C03654=1194.031,57.850,-47.386,-179.235,5.821,148.807
C03655=1194.026,58.099,-47.403,-179.232,5.823,148.806
C03656=1194.021,58.349,-47.419,-179.230,5.824,148.805
C03657=1194.016,58.598,-47.436,-179.227,5.824,148.805
C03658=1194.011,58.848,-47.452,-179.225,5.825,148.804
C03659=1194.006,59.097,-47.468,-179.223,5.826,148.804
C03660=1194.001,59.346,-47.485,-179.219,5.827,148.803
C03661=1193.997,59.596,-47.502,-179.217,5.828,148.803
C03662=1193.992,59.844,-47.518,-179.215,5.828,148.802
C03663=1193.986,60.095,-47.535,-179.212,5.829,148.801
C03664=1193.981,60.344,-47.551,-179.209,5.831,148.801
C03665=1193.976,60.593,-47.568,-179.207,5.831,148.800
C03666=1193.972,60.843,-47.584,-179.204,5.832,148.800
C03667=1193.966,61.092,-47.601,-179.202,5.833,148.799
C03668=1193.962,61.341,-47.618,-179.199,5.833,148.798
C03669=1193.957,61.591,-47.634,-179.196,5.834,148.798
C03670=1193.952,61.840,-47.650,-179.194,5.835,148.797
C03671=1193.947,62.090,-47.667,-179.191,5.836,148.797
C03672=1193.942,62.339,-47.684,-179.189,5.836,148.796
C03673=1193.937,62.588,-47.700,-179.186,5.838,148.796
C03674=1193.932,62.838,-47.718,-179.183,5.839,148.795
C03675=1193.927,63.087,-47.734,-179.181,5.840,148.794
C03676=1193.922,63.336,-47.751,-179.178,5.840,148.794
C03677=1193.918,63.586,-47.767,-179.176,5.841,148.793
C03678=1193.913,63.836,-47.784,-179.173,5.842,148.793
C03679=1193.907,64.084,-47.801,-179.170,5.843,148.792
C03680=1193.903,64.334,-47.817,-179.168,5.843,148.791
C03681=1193.897,64.584,-47.834,-179.166,5.844,148.791
C03682=1193.892,64.833,-47.850,-179.162,5.846,148.790
C03683=1193.887,65.083,-47.868,-179.160,5.847,148.790
C03684=1193.883,65.332,-47.884,-179.158,5.847,148.789
C03685=1193.878,65.581,-47.901,-179.155,5.848,148.789
C03686=1193.872,65.831,-47.918,-179.152,5.849,148.788
C03687=1193.868,66.080,-47.934,-179.150,5.850,148.787
C03688=1193.864,66.329,-47.952,-179.147,5.851,148.787
C03689=1193.858,66.578,-47.969,-179.145,5.851,148.786
C03690=1193.853,66.828,-47.985,-179.142,5.853,148.786
C03691=1193.848,67.078,-48.003,-179.140,5.854,148.785
C03692=1193.843,67.326,-48.019,-179.137,5.854,148.785
C03693=1193.839,67.576,-48.036,-179.134,5.855,148.784
C03694=1193.833,67.826,-48.053,-179.132,5.856,148.784
C03695=1193.829,68.075,-48.070,-179.129,5.857,148.783
C03696=1193.823,68.324,-48.086,-179.126,5.858,148.782
C03697=1193.819,68.574,-48.103,-179.124,5.858,148.782
C03698=1193.813,68.823,-48.120,-179.121,5.860,148.781
C03699=1193.809,69.072,-48.138,-179.119,5.861,148.781
C03700=1193.804,69.322,-48.155,-179.116,5.861,148.780
C03701=1193.799,69.571,-48.171,-179.113,5.863,148.779
C03702=1193.794,69.820,-48.188,-179.111,5.864,148.779
C03703=1193.789,70.070,-48.205,-179.108,5.864,148.778
C03704=1193.785,70.320,-48.222,-179.106,5.865,148.778
C03705=1193.779,70.568,-48.240,-179.103,5.866,148.777
C03706=1193.775,70.818,-48.256,-179.100,5.867,148.777
C03707=1193.770,71.067,-48.274,-179.098,5.868,148.776
C03708=1193.765,71.317,-48.290,-179.095,5.868,148.775
C03709=1193.760,71.567,-48.307,-179.093,5.870,148.775
C03710=1193.754,71.815,-48.325,-179.090,5.871,148.774
C03711=1193.750,72.065,-48.342,-179.087,5.871,148.774
C03712=1193.745,72.314,-48.359,-179.085,5.873,148.773
C03713=1193.740,72.564,-48.376,-179.082,5.873,148.773
C03714=1193.735,72.813,-48.394,-179.080,5.874,148.772
C03715=1193.731,73.063,-48.410,-179.077,5.875,148.771
C03716=1193.725,73.312,-48.427,-179.074,5.876,148.771
C03717=1193.721,73.561,-48.445,-179.072,5.877,148.770
C03718=1193.716,73.810,-48.462,-179.069,5.878,148.770
C03719=1193.710,74.060,-48.479,-179.067,5.879,148.769
C03720=1193.706,74.310,-48.496,-179.064,5.880,148.769
C03721=1193.701,74.559,-48.514,-179.061,5.880,148.768
C03722=1193.696,74.808,-48.530,-179.059,5.882,148.768
C03723=1193.691,75.057,-48.548,-179.056,5.883,148.767
C03724=1193.686,75.307,-48.565,-179.054,5.884,148.766
C03725=1193.681,75.556,-48.582,-179.051,5.884,148.766
C03726=1193.676,75.805,-48.600,-179.049,5.886,148.765
C03727=1193.671,76.055,-48.617,-179.046,5.886,148.765
C03728=1193.667,76.305,-48.634,-179.043,5.887,148.764
C03729=1193.662,76.554,-48.652,-179.041,5.889,148.764
C03730=1193.657,76.802,-48.668,-179.038,5.889,148.763
C03731=1193.652,77.052,-48.686,-179.036,5.890,148.763
C03732=1193.647,77.301,-48.703,-179.033,5.892,148.762
C03733=1193.642,77.550,-48.721,-179.030,5.892,148.762
C03734=1193.637,77.800,-48.738,-179.028,5.893,148.761
C03735=1193.632,78.049,-48.756,-179.025,5.894,148.760
C03736=1193.627,78.299,-48.773,-179.022,5.895,148.760
C03737=1193.623,78.549,-48.790,-179.020,5.896,148.759
C03738=1193.618,78.798,-48.808,-179.018,5.897,148.759
C03739=1193.612,79.048,-48.825,-179.014,5.898,148.758
C03740=1193.608,79.296,-48.843,-179.012,5.899,148.758
C03741=1193.602,79.545,-48.860,-179.010,5.900,148.757
C03742=1193.597,79.795,-48.878,-179.007,5.901,148.756
C03743=1193.593,80.044,-48.895,-179.004,5.902,148.756
C03744=1193.588,80.293,-48.912,-179.002,5.902,148.755
C03745=1193.583,80.562,-48.932,-178.999,5.904,148.755
C03746=1193.578,80.830,-48.950,-178.996,5.905,148.754
C03747=1193.572,81.099,-48.969,-178.993,5.906,148.754
C03748=1193.567,81.367,-48.988,-178.990,5.907,148.753
C03749=1193.562,81.616,-49.006,-178.988,5.908,148.752
C03750=1193.557,81.866,-49.023,-178.985,5.909,148.752
C03751=1193.552,82.115,-49.041,-178.983,5.911,148.751
C03752=1193.547,82.365,-49.058,-178.980,5.911,148.751
C03753=1193.542,82.614,-49.076,-178.977,5.912,148.750
C03754=1193.537,82.863,-49.094,-178.975,5.913,148.750
C03755=1193.533,83.112,-49.111,-178.972,5.914,148.749
C03756=1193.528,83.362,-49.129,-178.970,5.915,148.749
C03757=1193.523,83.611,-49.146,-178.967,5.916,148.748
C03758=1193.518,83.860,-49.164,-178.964,5.917,148.747
C03759=1193.513,84.110,-49.182,-178.962,5.918,148.747
C03760=1193.508,84.359,-49.200,-178.959,5.920,148.746
C03761=1193.503,84.608,-49.216,-178.957,5.920,148.746
C03762=1193.498,84.857,-49.234,-178.954,5.921,148.745
C03763=1193.494,85.107,-49.252,-178.951,5.922,148.745
C03764=1193.489,85.356,-49.270,-178.949,5.923,148.744
C03765=1193.483,85.606,-49.288,-178.946,5.925,148.744
C03766=1193.479,85.856,-49.306,-178.943,5.925,148.743
C03767=1193.474,86.105,-49.324,-178.941,5.926,148.743
C03768=1193.469,86.354,-49.342,-178.938,5.927,148.742
C03769=1193.464,86.603,-49.360,-178.936,5.928,148.741
C03770=1193.460,86.853,-49.377,-178.933,5.929,148.741
C03771=1193.455,87.102,-49.395,-178.930,5.931,148.740
C03772=1193.450,87.351,-49.412,-178.928,5.931,148.740
C03773=1193.445,87.600,-49.430,-178.926,5.932,148.739
C03774=1193.440,87.849,-49.448,-178.922,5.934,148.739
C03775=1193.435,88.099,-49.466,-178.920,5.934,148.738
C03776=1193.430,88.348,-49.484,-178.917,5.936,148.738
C03777=1193.425,88.597,-49.502,-178.915,5.937,148.737
C03778=1193.420,88.847,-49.520,-178.912,5.937,148.737
C03779=1193.415,89.096,-49.538,-178.909,5.939,148.736
C03780=1193.411,89.346,-49.556,-178.907,5.940,148.735
C03781=1193.406,89.595,-49.574,-178.904,5.941,148.735
C03782=1193.401,89.844,-49.592,-178.902,5.942,148.734
C03783=1193.396,90.093,-49.610,-178.899,5.942,148.734
C03784=1193.391,90.343,-49.627,-178.896,5.944,148.733
C03785=1193.386,90.592,-49.645,-178.894,5.945,148.733
C03786=1193.381,90.841,-49.663,-178.892,5.946,148.732
C03787=1193.376,91.090,-49.681,-178.888,5.947,148.732
C03788=1193.372,91.340,-49.699,-178.886,5.948,148.731
C03789=1193.367,91.590,-49.717,-178.883,5.949,148.731
C03790=1193.362,91.839,-49.735,-178.881,5.950,148.730
C03791=1193.357,92.088,-49.753,-178.878,5.951,148.729
C03792=1193.352,92.337,-49.771,-178.876,5.953,148.729
C03793=1193.348,92.586,-49.789,-178.873,5.953,148.728
C03794=1193.343,92.835,-49.807,-178.870,5.955,148.728
C03795=1193.338,93.086,-49.826,-178.868,5.955,148.727
C03796=1193.333,93.335,-49.844,-178.865,5.957,148.727
C03797=1193.328,93.584,-49.862,-178.862,5.958,148.726
C03798=1193.323,93.833,-49.880,-178.860,5.959,148.726
C03799=1193.318,94.082,-49.899,-178.857,5.960,148.725
C03800=1193.313,94.331,-49.917,-178.855,5.961,148.725
C03801=1193.309,94.581,-49.935,-178.852,5.962,148.724
C03802=1193.304,94.830,-49.953,-178.850,5.963,148.724
C03803=1193.299,95.079,-49.971,-178.847,5.964,148.723
C03804=1193.294,95.329,-49.990,-178.844,5.966,148.723
C03805=1193.289,95.578,-50.008,-178.842,5.966,148.722
C03806=1193.284,95.828,-50.026,-178.839,5.968,148.722
C03807=1193.279,96.077,-50.044,-178.836,5.968,148.721
C03808=1193.275,96.325,-50.063,-178.834,5.970,148.721
C03809=1193.270,96.575,-50.081,-178.831,5.971,148.720
C03810=1193.265,96.825,-50.100,-178.829,5.972,148.719
C03811=1193.260,97.074,-50.118,-178.826,5.973,148.719
C03812=1193.255,97.323,-50.136,-178.823,5.974,148.718
C03813=1193.250,97.572,-50.154,-178.820,5.975,148.718
C03814=1193.245,97.821,-50.172,-178.818,5.976,148.717
C03815=1193.240,98.071,-50.191,-178.815,5.978,148.717
C03816=1193.236,98.320,-50.209,-178.813,5.979,148.716
C03817=1193.231,98.569,-50.227,-178.810,5.980,148.716
C03818=1193.227,98.819,-50.246,-178.807,5.981,148.715
C03819=1193.222,99.068,-50.264,-178.805,5.982,148.715
C03820=1193.216,99.317,-50.283,-178.802,5.983,148.714
C03821=1193.211,99.566,-50.301,-178.800,5.984,148.714
C03822=1193.207,99.816,-50.320,-178.797,5.985,148.713
C03823=1193.201,100.065,-50.338,-178.795,5.986,148.713
C03824=1193.197,100.314,-50.356,-178.791,5.988,148.712
C03825=1193.192,100.563,-50.375,-178.789,5.989,148.712
C03826=1193.188,100.813,-50.393,-178.786,5.990,148.711
C03827=1193.182,101.062,-50.412,-178.784,5.991,148.711
C03828=1193.177,101.311,-50.431,-178.781,5.992,148.710
C03829=1193.173,101.561,-50.449,-178.779,5.993,148.710
C03830=1193.167,101.810,-50.468,-178.776,5.994,148.709
C03831=1193.163,102.059,-50.486,-178.773,5.996,148.709
C03832=1193.159,102.309,-50.505,-178.771,5.997,148.708
C03833=1193.153,102.557,-50.524,-178.768,5.998,148.707
C03834=1193.148,102.807,-50.542,-178.766,5.999,148.707
C03835=1193.144,103.057,-50.560,-178.763,6.000,148.706
C03836=1193.139,103.305,-50.580,-178.761,6.001,148.706
C03837=1193.134,103.555,-50.598,-178.757,6.003,148.705
C03838=1193.130,103.804,-50.617,-178.755,6.003,148.705
C03839=1193.124,104.053,-50.635,-178.752,6.005,148.704
C03840=1193.119,104.302,-50.654,-178.750,6.006,148.704
C03841=1193.115,104.552,-50.672,-178.747,6.007,148.703
C03842=1193.110,104.801,-50.692,-178.745,6.008,148.703
C03843=1193.105,105.050,-50.710,-178.742,6.010,148.702
C03844=1193.100,105.299,-50.729,-178.739,6.010,148.702
C03845=1193.095,105.549,-50.747,-178.737,6.012,148.701
C03846=1193.091,105.798,-50.766,-178.734,6.013,148.701
C03847=1193.086,106.047,-50.785,-178.731,6.015,148.700
C03848=1193.081,106.296,-50.804,-178.729,6.015,148.700
C03849=1193.076,106.565,-50.824,-178.726,6.017,148.699
C03850=1193.070,106.833,-50.845,-178.723,6.017,148.699
C03851=1193.065,107.101,-50.864,-178.720,6.019,148.698
C03852=1193.060,107.370,-50.885,-178.717,6.021,148.698
C03853=1193.055,107.619,-50.903,-178.715,6.021,148.697
C03854=1193.051,107.869,-50.923,-178.712,6.023,148.697
C03855=1193.046,108.118,-50.941,-178.710,6.024,148.696
C03856=1193.040,108.367,-50.960,-178.707,6.025,148.696
C03857=1193.036,108.616,-50.979,-178.705,6.026,148.695
C03858=1193.031,108.865,-50.998,-178.702,6.028,148.694
C03859=1193.027,109.115,-51.017,-178.699,6.028,148.694
C03860=1193.021,109.364,-51.036,-178.696,6.030,148.693
C03861=1193.017,109.613,-51.054,-178.694,6.031,148.693
C03862=1193.012,109.862,-51.074,-178.691,6.033,148.693
C03863=1193.008,110.112,-51.093,-178.689,6.033,148.692
C03864=1193.002,110.361,-51.111,-178.686,6.035,148.692
C03865=1192.997,110.610,-51.131,-178.683,6.035,148.691
C03866=1192.993,110.859,-51.150,-178.681,6.037,148.691
C03867=1192.987,111.108,-51.169,-178.679,6.038,148.690
C03868=1192.983,111.358,-51.187,-178.675,6.039,148.689
C03869=1192.978,111.607,-51.207,-178.673,6.040,148.689
C03870=1192.974,111.856,-51.226,-178.670,6.042,148.688
C03871=1192.968,112.105,-51.245,-178.667,6.044,148.688
C03872=1192.963,112.355,-51.264,-178.665,6.044,148.688
C03873=1192.959,112.604,-51.283,-178.662,6.046,148.687
C03874=1192.954,112.853,-51.302,-178.660,6.047,148.687
C03875=1192.949,113.102,-51.321,-178.657,6.048,148.686
C03876=1192.945,113.351,-51.341,-178.655,6.049,148.686
C03877=1192.939,113.601,-51.359,-178.652,6.051,148.685
C03878=1192.935,113.850,-51.378,-178.649,6.051,148.684
C03879=1192.930,114.099,-51.397,-178.647,6.053,148.684
C03880=1192.925,114.349,-51.417,-178.644,6.054,148.683
C03881=1192.920,114.597,-51.436,-178.641,6.056,148.683
C03882=1192.915,114.847,-51.455,-178.639,6.056,148.683
C03883=1192.911,115.096,-51.475,-178.636,6.058,148.682
C03884=1192.906,115.345,-51.493,-178.633,6.060,148.682
C03885=1192.901,115.595,-51.513,-178.631,6.060,148.681
C03886=1192.896,115.844,-51.532,-178.628,6.062,148.681
C03887=1192.892,116.093,-51.551,-178.626,6.063,148.680
C03888=1192.886,116.342,-51.570,-178.623,6.064,148.680
C03889=1192.882,116.592,-51.590,-178.621,6.065,148.679
C03890=1192.876,116.840,-51.609,-178.617,6.067,148.678
C03891=1192.872,117.090,-51.628,-178.615,6.068,148.678
C03892=1192.868,117.339,-51.648,-178.613,6.069,148.678
C03893=1192.862,117.588,-51.667,-178.609,6.071,148.677
C03894=1192.857,117.838,-51.687,-178.607,6.072,148.677
C03895=1192.853,118.086,-51.706,-178.605,6.073,148.676
C03896=1192.848,118.336,-51.725,-178.602,6.074,148.676
C03897=1192.843,118.585,-51.745,-178.599,6.076,148.675
C03898=1192.838,118.834,-51.764,-178.597,6.076,148.675
C03899=1192.834,119.084,-51.783,-178.594,6.078,148.674
C03900=1192.829,119.332,-51.803,-178.591,6.080,148.674
C03901=1192.824,119.582,-51.822,-178.589,6.080,148.673
C03902=1192.819,119.832,-51.842,-178.586,6.082,148.673
C03903=1192.814,120.080,-51.861,-178.584,6.083,148.672
C03904=1192.810,120.329,-51.881,-178.581,6.085,148.672
C03905=1192.805,120.579,-51.901,-178.578,6.085,148.671
C03906=1192.800,120.827,-51.920,-178.576,6.087,148.671
C03907=1192.795,121.077,-51.940,-178.573,6.089,148.670
C03908=1192.791,121.327,-51.959,-178.570,6.090,148.670
C03909=1192.785,121.575,-51.979,-178.568,6.091,148.669
C03910=1192.781,121.825,-51.998,-178.565,6.092,148.669
C03911=1192.776,122.073,-52.018,-178.562,6.094,148.668
C03912=1192.771,122.323,-52.037,-178.559,6.095,148.668
C03913=1192.767,122.572,-52.057,-178.557,6.096,148.667
C03914=1192.762,122.822,-52.077,-178.554,6.098,148.667
C03915=1192.757,123.071,-52.096,-178.552,6.098,148.666
C03916=1192.752,123.319,-52.116,-178.549,6.100,148.666
C03917=1192.747,123.569,-52.136,-178.546,6.102,148.666
C03918=1192.743,123.818,-52.155,-178.544,6.102,148.665
C03919=1192.738,124.067,-52.174,-178.541,6.104,148.665
C03920=1192.733,124.317,-52.194,-178.539,6.105,148.664
C03921=1192.728,124.565,-52.214,-178.536,6.107,148.664
C03922=1192.724,124.815,-52.234,-178.533,6.108,148.663
C03923=1192.719,125.064,-52.253,-178.531,6.109,148.663
C03924=1192.714,125.313,-52.274,-178.528,6.111,148.662
C03925=1192.709,125.562,-52.293,-178.526,6.112,148.662
C03926=1192.704,125.812,-52.313,-178.523,6.113,148.661
C03927=1192.700,126.060,-52.333,-178.520,6.115,148.661
C03928=1192.695,126.310,-52.353,-178.518,6.116,148.660
C03929=1192.690,126.559,-52.372,-178.515,6.117,148.660
C03930=1192.685,126.808,-52.392,-178.512,6.118,148.659
C03931=1192.681,127.057,-52.412,-178.510,6.120,148.659
C03932=1192.676,127.307,-52.432,-178.507,6.122,148.658
C03933=1192.671,127.555,-52.452,-178.504,6.122,148.658
C03934=1192.666,127.805,-52.471,-178.502,6.124,148.657
C03935=1192.662,128.054,-52.492,-178.499,6.126,148.657
C03936=1192.657,128.303,-52.511,-178.496,6.126,148.656
C03937=1192.652,128.552,-52.531,-178.494,6.128,148.656
C03938=1192.647,128.801,-52.551,-178.491,6.130,148.656
C03939=1192.642,129.051,-52.571,-178.489,6.131,148.655
C03940=1192.638,129.300,-52.591,-178.486,6.132,148.655
C03941=1192.633,129.549,-52.611,-178.484,6.133,148.654
C03942=1192.628,129.797,-52.631,-178.481,6.135,148.654
C03943=1192.623,130.047,-52.650,-178.478,6.136,148.653
C03944=1192.619,130.296,-52.671,-178.476,6.137,148.653
C03945=1192.613,130.546,-52.691,-178.473,6.139,148.652
C03946=1192.609,130.795,-52.711,-178.470,6.140,148.652
C03947=1192.604,131.044,-52.731,-178.468,6.141,148.651
C03948=1192.599,131.293,-52.751,-178.465,6.143,148.651
C03949=1192.594,131.542,-52.771,-178.462,6.145,148.651
C03950=1192.590,131.791,-52.791,-178.460,6.145,148.650
C03951=1192.585,132.041,-52.811,-178.457,6.147,148.650
C03952=1192.581,132.290,-52.831,-178.454,6.149,148.649
C03953=1192.575,132.559,-52.853,-178.452,6.150,148.649
C03954=1192.570,132.827,-52.875,-178.449,6.151,148.648
C03955=1192.565,133.096,-52.896,-178.446,6.153,148.648
C03956=1192.560,133.364,-52.919,-178.443,6.154,148.647
C03957=1192.555,133.614,-52.938,-178.440,6.156,148.647
C03958=1192.550,133.862,-52.959,-178.438,6.157,148.646
C03959=1192.545,134.111,-52.979,-178.435,6.159,148.646
C03960=1192.541,134.360,-52.998,-178.432,6.160,148.645
C03961=1192.535,134.610,-53.019,-178.430,6.161,148.645
C03962=1192.531,134.858,-53.040,-178.427,6.163,148.644
C03963=1192.526,135.108,-53.059,-178.425,6.164,148.644
C03964=1192.522,135.357,-53.080,-178.422,6.165,148.644
C03965=1192.517,135.606,-53.100,-178.419,6.167,148.643
C03966=1192.512,135.856,-53.120,-178.417,6.169,148.643
C03967=1192.508,136.105,-53.141,-178.414,6.170,148.642
C03968=1192.503,136.354,-53.161,-178.411,6.171,148.642
C03969=1192.497,136.602,-53.182,-178.409,6.173,148.641
C03970=1192.493,136.851,-53.202,-178.406,6.174,148.641
C03971=1192.488,137.101,-53.222,-178.404,6.175,148.640
C03972=1192.484,137.350,-53.242,-178.401,6.177,148.640
C03973=1192.478,137.599,-53.263,-178.398,6.179,148.639
C03974=1192.474,137.848,-53.283,-178.396,6.180,148.639
C03975=1192.469,138.098,-53.303,-178.393,6.181,148.639
C03976=1192.464,138.347,-53.324,-178.390,6.183,148.638
C03977=1192.460,138.596,-53.344,-178.388,6.184,148.638
C03978=1192.455,138.845,-53.365,-178.385,6.185,148.637
C03979=1192.450,139.094,-53.386,-178.382,6.187,148.637
C03980=1192.446,139.343,-53.406,-178.380,6.188,148.636
C03981=1192.441,139.592,-53.426,-178.377,6.190,148.636
C03982=1192.436,139.841,-53.447,-178.374,6.191,148.635
C03983=1192.431,140.091,-53.467,-178.372,6.193,148.635
C03984=1192.427,140.340,-53.487,-178.369,6.194,148.634
C03985=1192.422,140.589,-53.508,-178.366,6.196,148.634
C03986=1192.417,140.838,-53.529,-178.364,6.197,148.634
C03987=1192.413,141.087,-53.549,-178.362,6.198,148.633
C03988=1192.408,141.336,-53.570,-178.358,6.200,148.633
C03989=1192.403,141.585,-53.590,-178.356,6.201,148.632
C03990=1192.398,141.834,-53.611,-178.353,6.203,148.632
C03991=1192.394,142.083,-53.632,-178.351,6.204,148.631
C03992=1192.388,142.332,-53.653,-178.348,6.206,148.631
C03993=1192.384,142.581,-53.673,-178.345,6.207,148.630
C03994=1192.380,142.830,-53.694,-178.342,6.209,148.630
C03995=1192.374,143.080,-53.714,-178.340,6.210,148.630
C03996=1192.370,143.329,-53.735,-178.338,6.212,148.629
C03997=1192.365,143.578,-53.756,-178.334,6.213,148.629
C03998=1192.360,143.827,-53.776,-178.332,6.214,148.628
C03999=1192.355,144.076,-53.797,-178.330,6.216,148.628
C04000=1192.351,144.325,-53.818,-178.327,6.218,148.628
C04001=1192.346,144.574,-53.839,-178.324,6.219,148.627
C04002=1192.342,144.823,-53.860,-178.322,6.220,148.627
C04003=1192.337,145.073,-53.881,-178.319,6.222,148.626
C04004=1192.332,145.321,-53.901,-178.316,6.224,148.626
C04005=1192.327,145.571,-53.922,-178.314,6.225,148.625
C04006=1192.323,145.820,-53.943,-178.311,6.226,148.625
C04007=1192.318,146.069,-53.964,-178.308,6.228,148.624
C04008=1192.313,146.318,-53.984,-178.306,6.230,148.624
C04009=1192.308,146.567,-54.006,-178.303,6.231,148.624
C04010=1192.304,146.815,-54.026,-178.301,6.232,148.623
C04011=1192.299,147.065,-54.047,-178.298,6.234,148.623
C04012=1192.294,147.314,-54.067,-178.295,6.235,148.622
C04013=1192.290,147.564,-54.089,-178.292,6.237,148.622
C04014=1192.285,147.812,-54.110,-178.290,6.238,148.621
C04015=1192.280,148.061,-54.131,-178.288,6.240,148.621
C04016=1192.275,148.311,-54.152,-178.284,6.241,148.620
C04017=1192.271,148.559,-54.172,-178.282,6.243,148.620
C04018=1192.266,148.808,-54.194,-178.280,6.244,148.620
C04019=1192.261,149.057,-54.215,-178.277,6.246,148.619
C04020=1192.257,149.307,-54.235,-178.274,6.248,148.619
C04021=1192.252,149.556,-54.256,-178.272,6.249,148.619
C04022=1192.247,149.805,-54.278,-178.268,6.251,148.618
C04023=1192.242,150.054,-54.299,-178.266,6.252,148.618
C04024=1192.237,150.303,-54.319,-178.264,6.254,148.617
C04025=1192.232,150.552,-54.341,-178.261,6.255,148.617
C04026=1192.229,150.801,-54.362,-178.258,6.257,148.616
C04027=1192.223,151.051,-54.383,-178.256,6.258,148.616
C04028=1192.218,151.299,-54.405,-178.253,6.260,148.615
C04029=1192.214,151.548,-54.425,-178.250,6.261,148.615
C04030=1192.209,151.797,-54.447,-178.248,6.263,148.615
C04031=1192.204,152.046,-54.468,-178.245,6.265,148.614
C04032=1192.200,152.296,-54.488,-178.243,6.266,148.614
C04033=1192.195,152.544,-54.510,-178.240,6.267,148.613
C04034=1192.190,152.794,-54.531,-178.237,6.269,148.613
C04035=1192.185,153.042,-54.553,-178.234,6.271,148.613
C04036=1192.181,153.292,-54.573,-178.232,6.273,148.612
C04037=1192.177,153.541,-54.595,-178.229,6.274,148.612
C04038=1192.171,153.790,-54.616,-178.227,6.275,148.611
C04039=1192.166,154.039,-54.638,-178.224,6.277,148.611
C04040=1192.162,154.287,-54.658,-178.221,6.279,148.610
C04041=1192.158,154.537,-54.680,-178.218,6.280,148.610
C04042=1192.153,154.786,-54.701,-178.216,6.281,148.610
C04043=1192.148,155.035,-54.723,-178.213,6.283,148.609
C04044=1192.143,155.284,-54.744,-178.211,6.285,148.609
C04045=1192.139,155.533,-54.765,-178.208,6.287,148.609
C04046=1192.134,155.782,-54.786,-178.205,6.288,148.608
C04047=1192.129,156.031,-54.808,-178.203,6.289,148.608
C04048=1192.124,156.281,-54.829,-178.200,6.291,148.607
C04049=1192.120,156.530,-54.851,-178.197,6.293,148.607
C04050=1192.115,156.778,-54.872,-178.195,6.294,148.606
C04051=1192.110,157.027,-54.893,-178.192,6.296,148.606
C04052=1192.106,157.276,-54.915,-178.190,6.297,148.606
C04053=1192.101,157.526,-54.936,-178.187,6.298,148.605
C04054=1192.096,157.774,-54.958,-178.184,6.300,148.605
C04055=1192.092,158.024,-54.980,-178.181,6.302,148.604
C04056=1192.086,158.273,-55.001,-178.179,6.304,148.604
C04057=1192.082,158.541,-55.024,-178.176,6.306,148.604
C04058=1192.077,158.811,-55.047,-178.173,6.307,148.603
C04059=1192.072,159.080,-55.070,-178.170,6.309,148.603
C04060=1192.067,159.349,-55.094,-178.168,6.311,148.602
C04061=1192.061,159.598,-55.115,-178.165,6.312,148.602
C04062=1192.057,159.846,-55.137,-178.162,6.314,148.602
C04063=1192.053,160.095,-55.158,-178.160,6.316,148.601
C04064=1192.048,160.345,-55.179,-178.157,6.317,148.601
C04065=1192.043,160.593,-55.201,-178.154,6.318,148.600
C04066=1192.039,160.843,-55.223,-178.152,6.320,148.600
C04067=1192.034,161.091,-55.245,-178.149,6.322,148.599
C04068=1192.030,161.341,-55.267,-178.146,6.324,148.599
C04069=1192.024,161.590,-55.288,-178.144,6.325,148.599
C04070=1192.020,161.839,-55.309,-178.141,6.327,148.598
C04071=1192.015,162.088,-55.332,-178.139,6.328,148.598
C04072=1192.010,162.337,-55.353,-178.136,6.330,148.598
C04073=1192.006,162.585,-55.375,-178.133,6.331,148.597
C04074=1192.001,162.835,-55.397,-178.130,6.333,148.597
C04075=1191.996,163.084,-55.418,-178.128,6.335,148.596
C04076=1191.992,163.333,-55.440,-178.125,6.337,148.596
C04077=1191.987,163.582,-55.462,-178.122,6.339,148.595
C04078=1191.983,163.831,-55.484,-178.120,6.340,148.595
C04079=1191.978,164.080,-55.505,-178.117,6.341,148.595
C04080=1191.973,164.328,-55.527,-178.115,6.343,148.594
C04081=1191.968,164.578,-55.550,-178.112,6.345,148.594
C04082=1191.963,164.827,-55.571,-178.109,6.347,148.594
C04083=1191.959,165.076,-55.593,-178.107,6.348,148.593
C04084=1191.954,165.325,-55.615,-178.104,6.350,148.593
C04085=1191.950,165.574,-55.637,-178.101,6.352,148.592
C04086=1191.945,165.823,-55.659,-178.099,6.353,148.592
C04087=1191.941,166.072,-55.681,-178.096,6.354,148.592
C04088=1191.936,166.321,-55.703,-178.093,6.356,148.591
C04089=1191.931,166.569,-55.724,-178.091,6.358,148.591
C04090=1191.927,166.819,-55.746,-178.088,6.360,148.590
C04091=1191.922,167.067,-55.768,-178.085,6.362,148.590
C04092=1191.917,167.317,-55.791,-178.083,6.363,148.590
C04093=1191.912,167.566,-55.812,-178.080,6.365,148.589
C04094=1191.908,167.815,-55.834,-178.077,6.367,148.589
C04095=1191.903,168.064,-55.856,-178.075,6.368,148.589
C04096=1191.898,168.313,-55.878,-178.073,6.370,148.588
C04097=1191.893,168.562,-55.900,-178.070,6.371,148.588
C04098=1191.889,168.811,-55.923,-178.067,6.373,148.587
C04099=1191.884,169.059,-55.945,-178.064,6.375,148.587
C04100=1191.880,169.309,-55.967,-178.061,6.376,148.587
C04101=1191.875,169.557,-55.989,-178.059,6.378,148.586
C04102=1191.870,169.807,-56.011,-178.056,6.380,148.586
C04103=1191.865,170.055,-56.033,-178.053,6.382,148.585
C04104=1191.861,170.305,-56.055,-178.051,6.384,148.585
C04105=1191.857,170.554,-56.078,-178.049,6.385,148.585
C04106=1191.851,170.802,-56.100,-178.046,6.386,148.584
C04107=1191.847,171.052,-56.122,-178.043,6.388,148.584
C04108=1191.842,171.300,-56.144,-178.041,6.390,148.584
C04109=1191.838,171.549,-56.166,-178.038,6.392,148.583
C04110=1191.832,171.798,-56.189,-178.035,6.394,148.583
C04111=1191.828,172.047,-56.211,-178.033,6.395,148.582
C04112=1191.823,172.296,-56.232,-178.030,6.397,148.582
C04113=1191.819,172.545,-56.255,-178.027,6.399,148.582
C04114=1191.814,172.794,-56.278,-178.025,6.401,148.581
C04115=1191.809,173.043,-56.300,-178.022,6.402,148.581
C04116=1191.805,173.292,-56.322,-178.019,6.404,148.581
C04117=1191.800,173.541,-56.345,-178.017,6.406,148.580
C04118=1191.796,173.790,-56.367,-178.015,6.407,148.580
C04119=1191.791,174.039,-56.389,-178.012,6.409,148.580
C04120=1191.786,174.288,-56.412,-178.009,6.411,148.579
C04121=1191.782,174.537,-56.434,-178.006,6.412,148.579
C04122=1191.776,174.785,-56.457,-178.004,6.414,148.578
C04123=1191.772,175.035,-56.479,-178.001,6.416,148.578
C04124=1191.768,175.284,-56.501,-177.998,6.418,148.578
C04125=1191.763,175.532,-56.524,-177.996,6.420,148.577
C04126=1191.758,175.782,-56.546,-177.993,6.421,148.577
C04127=1191.754,176.031,-56.569,-177.990,6.423,148.577
C04128=1191.749,176.280,-56.591,-177.988,6.425,148.576
C04129=1191.745,176.528,-56.614,-177.985,6.427,148.576
C04130=1191.739,176.777,-56.636,-177.982,6.429,148.576
C04131=1191.735,177.026,-56.659,-177.980,6.430,148.575
C04132=1191.730,177.276,-56.681,-177.977,6.432,148.575
C04133=1191.725,177.524,-56.703,-177.974,6.434,148.574
C04134=1191.721,177.773,-56.726,-177.972,6.436,148.574
C04135=1191.717,178.022,-56.749,-177.969,6.437,148.574
C04136=1191.712,178.271,-56.771,-177.966,6.439,148.573
C04137=1191.707,178.520,-56.794,-177.964,6.441,148.573
C04138=1191.703,178.769,-56.816,-177.961,6.443,148.573
C04139=1191.698,179.018,-56.840,-177.959,6.444,148.572
C04140=1191.693,179.267,-56.861,-177.956,6.446,148.572
C04141=1191.689,179.516,-56.885,-177.954,6.447,148.572
C04142=1191.684,179.765,-56.907,-177.951,6.449,148.571
C04143=1191.679,180.013,-56.930,-177.948,6.451,148.571
C04144=1191.675,180.262,-56.952,-177.946,6.453,148.571
C04145=1191.670,180.512,-56.975,-177.943,6.455,148.570
C04146=1191.666,180.760,-56.998,-177.940,6.456,148.570
C04147=1191.661,181.009,-57.021,-177.938,6.458,148.569
C04148=1191.656,181.258,-57.043,-177.935,6.460,148.569
C04149=1191.652,181.507,-57.066,-177.932,6.462,148.569
C04150=1191.647,181.756,-57.090,-177.930,6.464,148.568
C04151=1191.642,182.005,-57.111,-177.927,6.465,148.568
C04152=1191.638,182.254,-57.135,-177.924,6.467,148.568
C04153=1191.634,182.503,-57.157,-177.922,6.469,148.567
C04154=1191.629,182.752,-57.181,-177.919,6.471,148.567
C04155=1191.623,183.001,-57.203,-177.916,6.473,148.567
C04156=1191.619,183.249,-57.226,-177.914,6.474,148.566
C04157=1191.615,183.498,-57.249,-177.911,6.476,148.566
C04158=1191.611,183.747,-57.272,-177.908,6.478,148.566
C04159=1191.606,183.997,-57.295,-177.906,6.480,148.565
C04160=1191.600,184.245,-57.318,-177.903,6.482,148.565
C04161=1191.596,184.514,-57.342,-177.900,6.484,148.564
C04162=1191.590,184.784,-57.367,-177.897,6.486,148.564
C04163=1191.585,185.054,-57.392,-177.894,6.488,148.564
C04164=1191.581,185.323,-57.417,-177.892,6.490,148.563
C04165=1191.576,185.572,-57.440,-177.889,6.491,148.563
C04166=1191.571,185.822,-57.463,-177.886,6.493,148.563
C04167=1191.567,186.070,-57.486,-177.884,6.495,148.562
C04168=1191.563,186.319,-57.509,-177.881,6.497,148.562
C04169=1191.558,186.568,-57.533,-177.878,6.499,148.562
C04170=1191.553,186.816,-57.555,-177.876,6.500,148.561
C04171=1191.549,187.065,-57.578,-177.873,6.502,148.561
C04172=1191.544,187.314,-57.602,-177.870,6.504,148.561
C04173=1191.539,187.563,-57.625,-177.868,6.506,148.560
C04174=1191.535,187.812,-57.648,-177.865,6.508,148.560
C04175=1191.530,188.061,-57.671,-177.862,6.510,148.560
C04176=1191.526,188.310,-57.695,-177.860,6.512,148.559
C04177=1191.520,188.559,-57.718,-177.857,6.514,148.559
C04178=1191.517,188.807,-57.740,-177.854,6.516,148.559
C04179=1191.512,189.056,-57.764,-177.852,6.518,148.558
C04180=1191.507,189.305,-57.787,-177.849,6.519,148.558
C04181=1191.502,189.554,-57.811,-177.846,6.521,148.558
C04182=1191.498,189.803,-57.834,-177.844,6.523,148.557
C04183=1191.493,190.052,-57.857,-177.841,6.525,148.557
C04184=1191.489,190.301,-57.880,-177.838,6.527,148.557
C04185=1191.484,190.550,-57.903,-177.836,6.528,148.556
C04186=1191.479,190.798,-57.926,-177.833,6.530,148.556
C04187=1191.474,191.048,-57.950,-177.830,6.532,148.556
C04188=1191.470,191.297,-57.973,-177.828,6.534,148.555
C04189=1191.465,191.546,-57.996,-177.826,6.536,148.555
C04190=1191.461,191.794,-58.019,-177.823,6.538,148.555
C04191=1191.457,192.043,-58.043,-177.820,6.540,148.554
C04192=1191.452,192.292,-58.067,-177.818,6.541,148.554
C04193=1191.447,192.541,-58.090,-177.815,6.543,148.554
C04194=1191.443,192.790,-58.113,-177.812,6.545,148.553
C04195=1191.438,193.039,-58.137,-177.809,6.548,148.553
C04196=1191.433,193.288,-58.160,-177.806,6.549,148.553
C04197=1191.429,193.536,-58.184,-177.804,6.552,148.553
C04198=1191.424,193.785,-58.207,-177.801,6.553,148.552
C04199=1191.419,194.034,-58.231,-177.799,6.555,148.552
C04200=1191.415,194.283,-58.254,-177.796,6.557,148.551
C04201=1191.410,194.532,-58.278,-177.794,6.559,148.551
C04202=1191.406,194.781,-58.302,-177.791,6.561,148.551
C04203=1191.401,195.030,-58.325,-177.788,6.562,148.550
C04204=1191.396,195.279,-58.348,-177.786,6.564,148.550
C04205=1191.392,195.527,-58.372,-177.783,6.566,148.550
C04206=1191.387,195.776,-58.396,-177.781,6.568,148.550
C04207=1191.382,196.025,-58.419,-177.778,6.570,148.549
C04208=1191.378,196.274,-58.443,-177.775,6.573,148.549
C04209=1191.373,196.523,-58.467,-177.772,6.574,148.549
C04210=1191.369,196.772,-58.490,-177.769,6.576,148.548
C04211=1191.364,197.020,-58.514,-177.767,6.578,148.548
C04212=1191.359,197.269,-58.537,-177.764,6.580,148.548
C04213=1191.355,197.518,-58.561,-177.762,6.582,148.547
C04214=1191.350,197.767,-58.585,-177.759,6.584,148.547
C04215=1191.346,198.016,-58.608,-177.757,6.586,148.547
C04216=1191.341,198.264,-58.632,-177.754,6.587,148.546
C04217=1191.337,198.513,-58.656,-177.751,6.589,148.546
C04218=1191.332,198.762,-58.680,-177.748,6.592,148.546
C04219=1191.327,199.011,-58.703,-177.745,6.594,148.545
C04220=1191.323,199.259,-58.727,-177.743,6.596,148.545
C04221=1191.319,199.509,-58.751,-177.741,6.598,148.545
C04222=1191.315,199.757,-58.775,-177.738,6.599,148.545
C04223=1191.309,200.007,-58.799,-177.735,6.601,148.544
C04224=1191.305,200.255,-58.823,-177.733,6.603,148.544
C04225=1191.300,200.504,-58.846,-177.730,6.605,148.543
C04226=1191.296,200.752,-58.870,-177.728,6.607,148.543
C04227=1191.291,201.001,-58.894,-177.725,6.610,148.543
C04228=1191.287,201.250,-58.918,-177.722,6.611,148.543
C04229=1191.282,201.499,-58.941,-177.719,6.613,148.542
C04230=1191.277,201.748,-58.966,-177.717,6.615,148.542
C04231=1191.273,201.997,-58.990,-177.714,6.617,148.542
C04232=1191.268,202.246,-59.014,-177.712,6.619,148.542
C04233=1191.264,202.494,-59.038,-177.709,6.621,148.541
C04234=1191.259,202.743,-59.061,-177.706,6.622,148.541
C04235=1191.254,202.992,-59.086,-177.703,6.625,148.541
C04236=1191.250,203.240,-59.110,-177.701,6.627,148.540
C04237=1191.246,203.490,-59.134,-177.698,6.629,148.540
C04238=1191.241,203.739,-59.158,-177.696,6.631,148.540
C04239=1191.237,203.987,-59.182,-177.693,6.633,148.539
C04240=1191.231,204.236,-59.206,-177.690,6.635,148.539
C04241=1191.227,204.485,-59.230,-177.688,6.636,148.539
C04242=1191.223,204.733,-59.254,-177.685,6.639,148.538
C04243=1191.219,204.982,-59.278,-177.682,6.641,148.538
C04244=1191.213,205.232,-59.302,-177.680,6.643,148.538
C04245=1191.209,205.480,-59.326,-177.677,6.645,148.538
C04246=1191.204,205.728,-59.350,-177.674,6.647,148.537
C04247=1191.199,205.977,-59.375,-177.672,6.648,148.537
C04248=1191.195,206.227,-59.399,-177.669,6.651,148.537
C04249=1191.191,206.475,-59.423,-177.666,6.653,148.536
C04250=1191.186,206.724,-59.447,-177.664,6.655,148.536
C04251=1191.181,206.972,-59.472,-177.661,6.657,148.536
C04252=1191.177,207.221,-59.496,-177.658,6.659,148.535
C04253=1191.172,207.470,-59.521,-177.656,6.661,148.535
C04254=1191.168,207.719,-59.544,-177.654,6.662,148.535
C04255=1191.163,207.968,-59.568,-177.650,6.665,148.535
C04256=1191.158,208.216,-59.593,-177.648,6.667,148.534
C04257=1191.154,208.466,-59.617,-177.645,6.669,148.534
C04258=1191.149,208.714,-59.642,-177.643,6.671,148.534
C04259=1191.145,208.963,-59.666,-177.640,6.673,148.534
C04260=1191.140,209.211,-59.690,-177.637,6.675,148.533
C04261=1191.136,209.460,-59.715,-177.634,6.677,148.533
C04262=1191.132,209.709,-59.739,-177.632,6.679,148.533
C04263=1191.126,209.958,-59.764,-177.629,6.681,148.532
C04264=1191.123,210.207,-59.788,-177.627,6.683,148.532
C04265=1191.117,210.478,-59.814,-177.624,6.686,148.532
C04266=1191.112,210.748,-59.841,-177.621,6.687,148.531
C04267=1191.107,211.018,-59.868,-177.618,6.690,148.531
C04268=1191.103,211.288,-59.894,-177.615,6.692,148.531
C04269=1191.098,211.537,-59.919,-177.613,6.694,148.531
C04270=1191.094,211.786,-59.943,-177.610,6.696,148.530
C04271=1191.089,212.035,-59.968,-177.607,6.698,148.530
C04272=1191.085,212.283,-59.992,-177.604,6.700,148.530
C04273=1191.079,212.532,-60.017,-177.602,6.702,148.530
C04274=1191.076,212.781,-60.041,-177.600,6.704,148.529
C04275=1191.071,213.030,-60.066,-177.597,6.706,148.529
C04276=1191.066,213.278,-60.090,-177.594,6.709,148.529
C04277=1191.062,213.527,-60.116,-177.592,6.711,148.529
C04278=1191.057,213.776,-60.140,-177.589,6.713,148.528
C04279=1191.052,214.024,-60.164,-177.586,6.714,148.528
C04280=1191.048,214.274,-60.189,-177.583,6.717,148.528
C04281=1191.043,214.522,-60.213,-177.581,6.719,148.527
C04282=1191.038,214.771,-60.238,-177.578,6.721,148.527
C04283=1191.035,215.019,-60.263,-177.576,6.723,148.527
C04284=1191.030,215.268,-60.288,-177.573,6.725,148.527
C04285=1191.025,215.518,-60.313,-177.570,6.728,148.526
C04286=1191.021,215.766,-60.337,-177.567,6.729,148.526
C04287=1191.016,216.014,-60.362,-177.565,6.731,148.526
C04288=1191.012,216.263,-60.387,-177.563,6.733,148.526
C04289=1191.007,216.512,-60.412,-177.559,6.736,148.525
C04290=1191.003,216.761,-60.437,-177.557,6.738,148.525
C04291=1190.998,217.009,-60.461,-177.554,6.740,148.525
C04292=1190.993,217.258,-60.486,-177.552,6.742,148.524
C04293=1190.989,217.507,-60.511,-177.549,6.744,148.524
C04294=1190.985,217.755,-60.536,-177.546,6.746,148.524
C04295=1190.980,218.004,-60.561,-177.544,6.748,148.524
C04296=1190.975,218.253,-60.586,-177.541,6.750,148.523
C04297=1190.972,218.502,-60.611,-177.539,6.752,148.523
C04298=1190.966,218.750,-60.635,-177.536,6.755,148.523
C04299=1190.961,218.999,-60.660,-177.533,6.757,148.523
C04300=1190.958,219.248,-60.685,-177.531,6.759,148.522
C04301=1190.953,219.496,-60.710,-177.528,6.760,148.522
C04302=1190.948,219.745,-60.736,-177.525,6.763,148.522
C04303=1190.943,219.994,-60.760,-177.523,6.765,148.522
C04304=1190.939,220.243,-60.785,-177.520,6.767,148.521
C04305=1190.935,220.491,-60.810,-177.518,6.769,148.521
C04306=1190.930,220.740,-60.835,-177.515,6.772,148.521
C04307=1190.925,220.989,-60.861,-177.512,6.774,148.520
C04308=1190.922,221.238,-60.885,-177.510,6.776,148.520
C04309=1190.917,221.486,-60.910,-177.507,6.778,148.520
C04310=1190.912,221.735,-60.935,-177.504,6.780,148.520
C04311=1190.907,221.983,-60.961,-177.502,6.782,148.520
C04312=1190.904,222.232,-60.985,-177.499,6.784,148.519
C04313=1190.899,222.481,-61.011,-177.496,6.786,148.519
C04314=1190.894,222.729,-61.036,-177.494,6.789,148.519
C04315=1190.889,222.978,-61.061,-177.491,6.791,148.519
C04316=1190.885,223.227,-61.087,-177.488,6.793,148.518
C04317=1190.881,223.476,-61.112,-177.486,6.795,148.518
C04318=1190.876,223.724,-61.137,-177.483,6.798,148.518
C04319=1190.872,223.973,-61.162,-177.480,6.799,148.517
C04320=1190.867,224.222,-61.187,-177.478,6.801,148.517
C04321=1190.863,224.470,-61.213,-177.475,6.803,148.517
C04322=1190.858,224.719,-61.237,-177.472,6.806,148.517
C04323=1190.854,224.968,-61.263,-177.470,6.808,148.517
C04324=1190.849,225.216,-61.289,-177.467,6.810,148.516
C04325=1190.844,225.465,-61.314,-177.464,6.813,148.516
C04326=1190.840,225.714,-61.339,-177.462,6.815,148.516
C04327=1190.835,225.962,-61.365,-177.459,6.817,148.516
C04328=1190.832,226.211,-61.390,-177.457,6.819,148.515
C04329=1190.827,226.460,-61.415,-177.454,6.821,148.515
C04330=1190.822,226.708,-61.440,-177.451,6.823,148.515
C04331=1190.818,226.957,-61.466,-177.449,6.825,148.515
C04332=1190.813,227.205,-61.491,-177.446,6.828,148.514
C04333=1190.809,227.455,-61.517,-177.443,6.830,148.514
C04334=1190.804,227.703,-61.542,-177.441,6.832,148.514
C04335=1190.800,227.952,-61.568,-177.439,6.834,148.514
C04336=1190.795,228.200,-61.593,-177.436,6.837,148.514
C04337=1190.791,228.449,-61.619,-177.433,6.839,148.513
C04338=1190.786,228.698,-61.644,-177.431,6.840,148.513
C04339=1190.782,228.947,-61.670,-177.428,6.843,148.513
C04340=1190.777,229.195,-61.695,-177.425,6.845,148.513
C04341=1190.773,229.444,-61.721,-177.423,6.847,148.512
C04342=1190.769,229.693,-61.746,-177.420,6.849,148.512
C04343=1190.764,229.941,-61.772,-177.417,6.852,148.512
C04344=1190.760,230.189,-61.798,-177.415,6.854,148.512
C04345=1190.755,230.438,-61.823,-177.412,6.856,148.511
C04346=1190.750,230.687,-61.849,-177.410,6.859,148.511
C04347=1190.746,230.935,-61.875,-177.407,6.861,148.511
C04348=1190.741,231.184,-61.901,-177.404,6.862,148.511
C04349=1190.736,231.433,-61.926,-177.402,6.865,148.511
C04350=1190.732,231.682,-61.951,-177.399,6.867,148.510
C04351=1190.728,231.931,-61.977,-177.397,6.869,148.510
C04352=1190.724,232.179,-62.003,-177.394,6.872,148.510
C04353=1190.719,232.427,-62.028,-177.391,6.874,148.510
C04354=1190.715,232.676,-62.055,-177.389,6.876,148.509
C04355=1190.710,232.925,-62.081,-177.386,6.879,148.509
C04356=1190.705,233.173,-62.106,-177.383,6.881,148.509
C04357=1190.701,233.422,-62.132,-177.381,6.883,148.509
C04358=1190.697,233.671,-62.158,-177.378,6.886,148.509
C04359=1190.692,233.919,-62.184,-177.375,6.887,148.508
C04360=1190.687,234.167,-62.209,-177.373,6.890,148.508
C04361=1190.683,234.417,-62.235,-177.371,6.891,148.508
C04362=1190.678,234.665,-62.261,-177.367,6.894,148.508
C04363=1190.674,234.914,-62.287,-177.365,6.896,148.508
C04364=1190.669,235.162,-62.312,-177.362,6.899,148.507
C04365=1190.665,235.410,-62.339,-177.360,6.901,148.507
C04366=1190.660,235.660,-62.365,-177.357,6.903,148.507
C04367=1190.656,235.908,-62.391,-177.354,6.906,148.507
C04368=1190.652,236.157,-62.417,-177.352,6.908,148.506
C04369=1190.647,236.428,-62.445,-177.349,6.911,148.506
C04370=1190.642,236.700,-62.473,-177.346,6.912,148.506
C04371=1190.637,236.972,-62.502,-177.343,6.915,148.506
C04372=1190.632,237.242,-62.530,-177.341,6.917,148.506
C04373=1190.628,237.491,-62.556,-177.338,6.920,148.505
C04374=1190.623,237.740,-62.582,-177.335,6.922,148.505
C04375=1190.619,237.989,-62.609,-177.332,6.925,148.505
C04376=1190.614,238.237,-62.634,-177.330,6.927,148.505
C04377=1190.610,238.486,-62.660,-177.328,6.929,148.505
C04378=1190.605,238.734,-62.687,-177.324,6.931,148.504
C04379=1190.601,238.983,-62.712,-177.322,6.934,148.504
C04380=1190.597,239.232,-62.738,-177.320,6.935,148.504
C04381=1190.592,239.480,-62.765,-177.317,6.938,148.504
C04382=1190.588,239.729,-62.791,-177.314,6.940,148.503
C04383=1190.583,239.978,-62.817,-177.312,6.942,148.503
C04384=1190.579,240.226,-62.844,-177.309,6.945,148.503
C04385=1190.574,240.474,-62.869,-177.307,6.947,148.503
C04386=1190.569,240.723,-62.896,-177.304,6.950,148.503
C04387=1190.565,240.972,-62.922,-177.301,6.952,148.503
C04388=1190.561,241.220,-62.948,-177.299,6.954,148.502
C04389=1190.556,241.469,-62.975,-177.296,6.957,148.502
C04390=1190.552,241.718,-63.001,-177.294,6.959,148.502
C04391=1190.547,241.966,-63.028,-177.291,6.962,148.502
C04392=1190.543,242.215,-63.053,-177.288,6.964,148.502
C04393=1190.538,242.463,-63.080,-177.286,6.966,148.501
C04394=1190.534,242.712,-63.106,-177.283,6.969,148.501
C04395=1190.529,242.960,-63.133,-177.280,6.970,148.501
C04396=1190.525,243.209,-63.159,-177.278,6.973,148.501
C04397=1190.521,243.457,-63.185,-177.275,6.975,148.501
C04398=1190.516,243.706,-63.212,-177.273,6.977,148.501
C04399=1190.512,243.954,-63.238,-177.270,6.980,148.500
C04400=1190.507,244.203,-63.265,-177.268,6.982,148.500
C04401=1190.503,244.452,-63.291,-177.265,6.984,148.500
C04402=1190.498,244.700,-63.318,-177.262,6.987,148.500
C04403=1190.494,244.949,-63.344,-177.260,6.989,148.499
C04404=1190.490,245.197,-63.371,-177.257,6.992,148.499
C04405=1190.486,245.446,-63.397,-177.255,6.994,148.499
C04406=1190.481,245.695,-63.423,-177.252,6.996,148.499
C04407=1190.476,245.943,-63.451,-177.249,6.999,148.499
C04408=1190.472,246.191,-63.477,-177.247,7.001,148.499
C04409=1190.467,246.441,-63.503,-177.244,7.004,148.499
C04410=1190.463,246.689,-63.530,-177.241,7.005,148.498
C04411=1190.459,246.937,-63.557,-177.239,7.008,148.498
C04412=1190.455,247.185,-63.583,-177.236,7.011,148.498
C04413=1190.450,247.435,-63.610,-177.234,7.012,148.498
C04414=1190.445,247.683,-63.637,-177.231,7.015,148.498
C04415=1190.441,247.931,-63.663,-177.228,7.017,148.497
C04416=1190.436,248.180,-63.690,-177.226,7.020,148.497
C04417=1190.431,248.429,-63.717,-177.223,7.022,148.497
C04418=1190.428,248.677,-63.743,-177.220,7.025,148.497
C04419=1190.423,248.925,-63.770,-177.218,7.027,148.497
C04420=1190.418,249.174,-63.797,-177.216,7.029,148.497
C04421=1190.414,249.422,-63.824,-177.213,7.032,148.497
C04422=1190.409,249.671,-63.850,-177.210,7.034,148.496
C04423=1190.405,249.920,-63.877,-177.207,7.037,148.496
C04424=1190.401,250.168,-63.904,-177.205,7.039,148.496
C04425=1190.396,250.416,-63.931,-177.202,7.042,148.496
C04426=1190.391,250.665,-63.958,-177.200,7.044,148.496
C04427=1190.388,250.913,-63.984,-177.197,7.046,148.495
C04428=1190.383,251.162,-64.011,-177.195,7.049,148.495
C04429=1190.378,251.410,-64.038,-177.192,7.051,148.495
C04430=1190.375,251.659,-64.065,-177.189,7.053,148.495
C04431=1190.370,251.908,-64.092,-177.187,7.056,148.495
C04432=1190.366,252.156,-64.119,-177.184,7.059,148.495
C04433=1190.361,252.404,-64.146,-177.182,7.060,148.494
C04434=1190.356,252.653,-64.173,-177.179,7.063,148.494
C04435=1190.352,252.901,-64.200,-177.176,7.065,148.494
C04436=1190.348,253.150,-64.227,-177.174,7.068,148.494
C04437=1190.343,253.398,-64.254,-177.171,7.070,148.494
C04438=1190.338,253.647,-64.281,-177.168,7.073,148.494
C04439=1190.335,253.896,-64.308,-177.166,7.075,148.494
C04440=1190.330,254.144,-64.335,-177.164,7.077,148.493
C04441=1190.326,254.393,-64.362,-177.161,7.080,148.493
C04442=1190.321,254.641,-64.389,-177.159,7.082,148.493
C04443=1190.316,254.890,-64.416,-177.156,7.085,148.493
C04444=1190.312,255.138,-64.443,-177.153,7.087,148.493
C04445=1190.308,255.387,-64.470,-177.150,7.090,148.493
C04446=1190.304,255.635,-64.497,-177.148,7.092,148.493
C04447=1190.299,255.883,-64.525,-177.145,7.095,148.492
C04448=1190.295,256.132,-64.552,-177.143,7.097,148.492
C04449=1190.290,256.380,-64.579,-177.140,7.100,148.492
C04450=1190.285,256.629,-64.606,-177.138,7.102,148.492
C04451=1190.281,256.878,-64.633,-177.135,7.105,148.492
C04452=1190.277,257.126,-64.660,-177.133,7.107,148.492
C04453=1190.272,257.374,-64.688,-177.129,7.110,148.491
C04454=1190.268,257.623,-64.715,-177.127,7.112,148.491
C04455=1190.264,257.871,-64.742,-177.125,7.115,148.491
C04456=1190.260,258.120,-64.769,-177.122,7.117,148.491
C04457=1190.255,258.368,-64.797,-177.119,7.120,148.491
C04458=1190.251,258.617,-64.824,-177.117,7.122,148.491
C04459=1190.246,258.865,-64.851,-177.114,7.124,148.491
C04460=1190.242,259.114,-64.879,-177.112,7.127,148.491
C04461=1190.238,259.362,-64.906,-177.109,7.130,148.490
C04462=1190.233,259.611,-64.933,-177.106,7.131,148.490
C04463=1190.229,259.859,-64.961,-177.104,7.134,148.490
C04464=1190.224,260.107,-64.988,-177.102,7.137,148.490
C04465=1190.220,260.356,-65.016,-177.098,7.139,148.490
C04466=1190.216,260.604,-65.043,-177.096,7.141,148.490
C04467=1190.211,260.853,-65.070,-177.093,7.144,148.490
C04468=1190.207,261.102,-65.098,-177.091,7.147,148.490
C04469=1190.203,261.350,-65.126,-177.088,7.149,148.489
C04470=1190.198,261.598,-65.153,-177.086,7.151,148.489
C04471=1190.194,261.846,-65.181,-177.083,7.154,148.489
C04472=1190.189,262.096,-65.209,-177.081,7.156,148.489
C04473=1190.184,262.368,-65.238,-177.078,7.159,148.489
C04474=1190.180,262.641,-65.269,-177.075,7.162,148.489
C04475=1190.174,262.914,-65.299,-177.072,7.165,148.488
C04476=1190.170,263.186,-65.329,-177.069,7.168,148.488
C04477=1190.165,263.435,-65.358,-177.066,7.171,148.488
C04478=1190.161,263.683,-65.385,-177.064,7.173,148.488
C04479=1190.156,263.931,-65.413,-177.061,7.176,148.488
C04480=1190.152,264.181,-65.440,-177.059,7.178,148.488
C04481=1190.148,264.428,-65.468,-177.056,7.181,148.488
C04482=1190.143,264.677,-65.495,-177.054,7.183,148.488
C04483=1190.139,264.926,-65.523,-177.051,7.186,148.488
C04484=1190.134,265.174,-65.551,-177.049,7.188,148.487
C04485=1190.130,265.423,-65.579,-177.046,7.191,148.487
C04486=1190.126,265.671,-65.607,-177.043,7.193,148.487
C04487=1190.121,265.919,-65.634,-177.041,7.196,148.487
C04488=1190.118,266.168,-65.662,-177.038,7.199,148.487
C04489=1190.113,266.416,-65.690,-177.036,7.201,148.487
C04490=1190.108,266.665,-65.717,-177.033,7.204,148.487
C04491=1190.104,266.913,-65.745,-177.030,7.206,148.487
C04492=1190.100,267.161,-65.773,-177.028,7.209,148.487
C04493=1190.095,267.410,-65.802,-177.026,7.211,148.486
C04494=1190.091,267.658,-65.829,-177.022,7.214,148.486
C04495=1190.086,267.906,-65.857,-177.020,7.217,148.486
C04496=1190.083,268.155,-65.885,-177.018,7.219,148.486
C04497=1190.077,268.403,-65.913,-177.015,7.222,148.486
C04498=1190.073,268.652,-65.941,-177.013,7.224,148.486
C04499=1190.069,268.900,-65.968,-177.009,7.227,148.486
C04500=1190.064,269.148,-65.997,-177.007,7.229,148.486
C04501=1190.060,269.397,-66.025,-177.005,7.232,148.486
C04502=1190.056,269.645,-66.053,-177.002,7.235,148.486
C04503=1190.051,269.894,-66.081,-176.999,7.237,148.485
C04504=1190.047,270.142,-66.108,-176.997,7.240,148.485
C04505=1190.043,270.391,-66.137,-176.994,7.242,148.485
C04506=1190.038,270.639,-66.165,-176.992,7.245,148.485
C04507=1190.034,270.887,-66.193,-176.989,7.247,148.485
C04508=1190.030,271.135,-66.221,-176.986,7.250,148.485
C04509=1190.025,271.384,-66.250,-176.984,7.253,148.485
C04510=1190.021,271.632,-66.277,-176.981,7.255,148.485
C04511=1190.017,271.880,-66.305,-176.979,7.258,148.485
C04512=1190.012,272.129,-66.334,-176.977,7.260,148.484
C04513=1190.008,272.377,-66.362,-176.974,7.263,148.484
C04514=1190.003,272.626,-66.390,-176.971,7.266,148.484
C04515=1189.999,272.874,-66.418,-176.968,7.268,148.484
C04516=1189.995,273.123,-66.446,-176.966,7.271,148.484
C04517=1189.991,273.371,-66.475,-176.964,7.273,148.484
C04518=1189.986,273.619,-66.503,-176.961,7.276,148.484
C04519=1189.982,273.868,-66.532,-176.958,7.279,148.484
C04520=1189.977,274.116,-66.559,-176.956,7.281,148.484
C04521=1189.973,274.364,-66.588,-176.953,7.284,148.484
C04522=1189.969,274.612,-66.616,-176.951,7.286,148.483
C04523=1189.964,274.861,-66.645,-176.948,7.289,148.483
C04524=1189.960,275.109,-66.672,-176.945,7.292,148.483
C04525=1189.955,275.358,-66.701,-176.943,7.294,148.483
C04526=1189.951,275.606,-66.729,-176.940,7.297,148.483
C04527=1189.946,275.855,-66.758,-176.937,7.300,148.483
C04528=1189.943,276.103,-66.787,-176.935,7.302,148.483
C04529=1189.938,276.351,-66.815,-176.932,7.305,148.483
C04530=1189.934,276.599,-66.843,-176.930,7.307,148.483
C04531=1189.929,276.848,-66.871,-176.927,7.310,148.483
C04532=1189.925,277.096,-66.900,-176.925,7.313,148.483
C04533=1189.920,277.344,-66.928,-176.922,7.315,148.482
C04534=1189.916,277.593,-66.957,-176.919,7.318,148.482
C04535=1189.912,277.841,-66.986,-176.917,7.321,148.482
C04536=1189.907,278.089,-67.014,-176.915,7.323,148.482
C04537=1189.903,278.338,-67.042,-176.912,7.326,148.482
C04538=1189.899,278.586,-67.072,-176.909,7.329,148.482
C04539=1189.895,278.834,-67.099,-176.907,7.331,148.482
C04540=1189.890,279.083,-67.128,-176.904,7.334,148.482
C04541=1189.886,279.331,-67.157,-176.902,7.336,148.482
C04542=1189.882,279.579,-67.185,-176.899,7.339,148.482
C04543=1189.877,279.828,-67.214,-176.896,7.342,148.482
C04544=1189.873,280.076,-67.243,-176.894,7.344,148.482
C04545=1189.869,280.324,-67.271,-176.891,7.347,148.482
C04546=1189.864,280.573,-67.300,-176.889,7.350,148.482
C04547=1189.860,280.821,-67.329,-176.886,7.352,148.482
C04548=1189.856,281.069,-67.357,-176.884,7.355,148.482
C04549=1189.852,281.318,-67.387,-176.881,7.358,148.481
C04550=1189.847,281.566,-67.415,-176.879,7.361,148.481
C04551=1189.843,281.814,-67.444,-176.876,7.363,148.481
C04552=1189.839,282.063,-67.473,-176.873,7.366,148.481
C04553=1189.834,282.311,-67.501,-176.871,7.368,148.481
C04554=1189.829,282.559,-67.530,-176.868,7.371,148.481
C04555=1189.826,282.808,-67.559,-176.865,7.374,148.481
C04556=1189.821,283.056,-67.588,-176.863,7.377,148.481
C04557=1189.816,283.304,-67.616,-176.860,7.380,148.481
C04558=1189.812,283.552,-67.646,-176.858,7.383,148.481
C04559=1189.809,283.800,-67.675,-176.856,7.385,148.481
C04560=1189.804,284.048,-67.703,-176.853,7.388,148.481
C04561=1189.799,284.297,-67.733,-176.850,7.391,148.481
C04562=1189.795,284.546,-67.761,-176.848,7.393,148.481
C04563=1189.791,284.794,-67.791,-176.845,7.396,148.481
C04564=1189.786,285.042,-67.819,-176.842,7.399,148.480
C04565=1189.782,285.290,-67.848,-176.840,7.401,148.480
C04566=1189.778,285.538,-67.877,-176.837,7.404,148.480
C04567=1189.774,285.787,-67.906,-176.835,7.407,148.480
C04568=1189.769,286.035,-67.935,-176.832,7.409,148.480
C04569=1189.765,286.283,-67.965,-176.830,7.412,148.480
C04570=1189.760,286.532,-67.993,-176.827,7.415,148.480
C04571=1189.756,286.780,-68.023,-176.825,7.417,148.480
C04572=1189.753,287.028,-68.052,-176.822,7.420,148.480
C04573=1189.747,287.276,-68.080,-176.819,7.423,148.480
C04574=1189.743,287.525,-68.110,-176.817,7.426,148.480
C04575=1189.739,287.773,-68.139,-176.815,7.428,148.480
C04576=1189.735,288.021,-68.168,-176.812,7.431,148.480
C04577=1189.730,288.295,-68.200,-176.809,7.434,148.480
C04578=1189.725,288.571,-68.233,-176.806,7.437,148.480
C04579=1189.721,288.845,-68.265,-176.804,7.440,148.480
C04580=1189.715,289.119,-68.297,-176.801,7.443,148.480
C04581=1189.711,289.368,-68.327,-176.798,7.446,148.479
C04582=1189.707,289.616,-68.356,-176.795,7.449,148.479
C04583=1189.703,289.864,-68.386,-176.793,7.451,148.479
C04584=1189.698,290.112,-68.415,-176.790,7.454,148.479
C04585=1189.694,290.361,-68.444,-176.787,7.457,148.479
C04586=1189.689,290.609,-68.473,-176.785,7.459,148.479
C04587=1189.685,290.857,-68.502,-176.783,7.462,148.479
C04588=1189.681,291.105,-68.532,-176.780,7.465,148.479
C04589=1189.677,291.354,-68.561,-176.777,7.468,148.479
C04590=1189.672,291.602,-68.591,-176.776,7.471,148.479
C04591=1189.668,291.850,-68.620,-176.773,7.474,148.479
C04592=1189.664,292.098,-68.650,-176.770,7.477,148.479
C04593=1189.660,292.347,-68.679,-176.767,7.480,148.479
C04594=1189.655,292.594,-68.708,-176.765,7.482,148.479
C04595=1189.651,292.842,-68.738,-176.763,7.485,148.479
C04596=1189.647,293.091,-68.767,-176.760,7.488,148.479
C04597=1189.643,293.339,-68.797,-176.758,7.490,148.479
C04598=1189.638,293.587,-68.826,-176.755,7.493,148.479
C04599=1189.634,293.836,-68.855,-176.752,7.496,148.479
C04600=1189.630,294.084,-68.885,-176.750,7.499,148.479
C04601=1189.625,294.332,-68.915,-176.747,7.501,148.479
C04602=1189.621,294.581,-68.944,-176.745,7.504,148.479
C04603=1189.617,294.829,-68.974,-176.742,7.507,148.479
C04604=1189.613,295.077,-69.004,-176.739,7.510,148.479
C04605=1189.609,295.325,-69.034,-176.737,7.513,148.479
C04606=1189.604,295.573,-69.063,-176.734,7.516,148.479
C04607=1189.600,295.821,-69.092,-176.732,7.519,148.479
C04608=1189.595,296.070,-69.122,-176.729,7.521,148.479
C04609=1189.591,296.318,-69.152,-176.727,7.524,148.479
C04610=1189.587,296.566,-69.182,-176.724,7.527,148.479
C04611=1189.583,296.814,-69.212,-176.721,7.530,148.479
C04612=1189.579,297.062,-69.241,-176.719,7.532,148.478
C04613=1189.574,297.311,-69.271,-176.717,7.535,148.479
C04614=1189.570,297.559,-69.300,-176.714,7.538,148.479
C04615=1189.566,297.807,-69.331,-176.712,7.541,148.479
C04616=1189.562,298.055,-69.360,-176.709,7.543,148.479
C04617=1189.557,298.304,-69.390,-176.707,7.546,148.479
C04618=1189.553,298.551,-69.420,-176.704,7.549,148.479
C04619=1189.549,298.800,-69.450,-176.701,7.552,148.478
C04620=1189.545,299.048,-69.479,-176.699,7.555,148.478
C04621=1189.540,299.296,-69.510,-176.696,7.558,148.478
C04622=1189.536,299.544,-69.539,-176.694,7.561,148.478
C04623=1189.532,299.792,-69.569,-176.691,7.564,148.478
C04624=1189.527,300.040,-69.600,-176.689,7.566,148.479
C04625=1189.523,300.289,-69.629,-176.687,7.569,148.478
C04626=1189.519,300.537,-69.659,-176.684,7.572,148.478
C04627=1189.514,300.785,-69.689,-176.681,7.575,148.478
C04628=1189.510,301.033,-69.719,-176.678,7.578,148.478
C04629=1189.506,301.281,-69.749,-176.676,7.580,148.478
C04630=1189.501,301.529,-69.779,-176.674,7.583,148.478
C04631=1189.497,301.777,-69.809,-176.671,7.586,148.478
C04632=1189.493,302.025,-69.839,-176.668,7.589,148.478
C04633=1189.489,302.274,-69.870,-176.666,7.592,148.478
C04634=1189.485,302.522,-69.899,-176.664,7.595,148.478
C04635=1189.480,302.770,-69.930,-176.661,7.598,148.478
C04636=1189.476,303.018,-69.959,-176.658,7.601,148.478
C04637=1189.471,303.266,-69.990,-176.656,7.603,148.478
C04638=1189.467,303.515,-70.020,-176.654,7.606,148.478
C04639=1189.463,303.762,-70.050,-176.651,7.609,148.478
C04640=1189.458,304.011,-70.080,-176.649,7.612,148.478
C04641=1189.455,304.259,-70.110,-176.646,7.615,148.478
C04642=1189.450,304.507,-70.140,-176.644,7.617,148.478
C04643=1189.446,304.755,-70.171,-176.641,7.620,148.478
C04644=1189.442,305.003,-70.201,-176.638,7.623,148.478
C04645=1189.438,305.252,-70.231,-176.636,7.626,148.478
C04646=1189.433,305.500,-70.262,-176.634,7.629,148.479
C04647=1189.429,305.747,-70.292,-176.631,7.632,148.479
C04648=1189.424,305.996,-70.322,-176.628,7.635,148.478
C04649=1189.421,306.244,-70.352,-176.626,7.638,148.478
C04650=1189.416,306.492,-70.383,-176.623,7.641,148.478
C04651=1189.412,306.740,-70.413,-176.621,7.643,148.479
C04652=1189.407,306.988,-70.443,-176.619,7.646,148.479
C04653=1189.403,307.236,-70.474,-176.616,7.650,148.479
C04654=1189.399,307.484,-70.504,-176.613,7.653,148.479
C04655=1189.395,307.733,-70.535,-176.611,7.656,148.479
C04656=1189.391,307.981,-70.565,-176.609,7.658,148.479
C04657=1189.386,308.229,-70.596,-176.606,7.661,148.479
C04658=1189.382,308.477,-70.626,-176.603,7.664,148.479
C04659=1189.378,308.724,-70.657,-176.601,7.667,148.479
C04660=1189.374,308.973,-70.688,-176.598,7.670,148.479
C04661=1189.370,309.221,-70.717,-176.596,7.673,148.479
C04662=1189.365,309.469,-70.748,-176.594,7.676,148.479
C04663=1189.360,309.717,-70.779,-176.591,7.679,148.479
C04664=1189.357,309.966,-70.809,-176.588,7.682,148.479
C04665=1189.352,310.214,-70.840,-176.586,7.685,148.479
C04666=1189.348,310.462,-70.871,-176.584,7.687,148.479
C04667=1189.344,310.709,-70.901,-176.581,7.690,148.479
C04668=1189.340,310.958,-70.932,-176.578,7.693,148.479
C04669=1189.335,311.206,-70.963,-176.576,7.696,148.479
C04670=1189.331,311.454,-70.993,-176.573,7.699,148.479
C04671=1189.327,311.702,-71.024,-176.571,7.702,148.479
C04672=1189.323,311.950,-71.055,-176.569,7.705,148.479
C04673=1189.319,312.198,-71.085,-176.566,7.708,148.479
C04674=1189.314,312.446,-71.116,-176.564,7.711,148.479
C04675=1189.310,312.694,-71.147,-176.561,7.714,148.479
C04676=1189.306,312.942,-71.178,-176.558,7.717,148.479
C04677=1189.302,313.190,-71.208,-176.557,7.719,148.479
C04678=1189.298,313.439,-71.239,-176.554,7.722,148.479
C04679=1189.293,313.687,-71.270,-176.551,7.725,148.479
C04680=1189.289,313.935,-71.300,-176.549,7.729,148.479
C04681=1189.284,314.211,-71.335,-176.546,7.732,148.479
C04682=1189.279,314.488,-71.369,-176.543,7.735,148.479
C04683=1189.275,314.764,-71.403,-176.540,7.739,148.480
C04684=1189.270,315.041,-71.439,-176.537,7.742,148.479
C04685=1189.266,315.288,-71.469,-176.535,7.745,148.480
C04686=1189.262,315.536,-71.500,-176.533,7.747,148.480
C04687=1189.258,315.785,-71.531,-176.530,7.750,148.480
C04688=1189.253,316.033,-71.561,-176.528,7.753,148.480
C04689=1189.249,316.280,-71.593,-176.525,7.756,148.480
C04690=1189.245,316.529,-71.624,-176.523,7.759,148.480
C04691=1189.240,316.777,-71.655,-176.520,7.763,148.480
C04692=1189.237,317.025,-71.685,-176.518,7.765,148.480
C04693=1189.232,317.273,-71.716,-176.516,7.768,148.480
C04694=1189.228,317.521,-71.748,-176.513,7.771,148.480
C04695=1189.224,317.769,-71.779,-176.511,7.774,148.480
C04696=1189.219,318.017,-71.809,-176.508,7.777,148.480
C04697=1189.216,318.265,-71.841,-176.506,7.781,148.480
C04698=1189.211,318.513,-71.872,-176.504,7.783,148.480
C04699=1189.206,318.761,-71.903,-176.501,7.786,148.480
C04700=1189.203,319.009,-71.935,-176.499,7.789,148.480
C04701=1189.198,319.257,-71.965,-176.496,7.792,148.480
C04702=1189.194,319.506,-71.997,-176.494,7.795,148.481
C04703=1189.190,319.753,-72.028,-176.491,7.798,148.481
C04704=1189.186,320.002,-72.059,-176.489,7.801,148.481
C04705=1189.181,320.249,-72.091,-176.487,7.804,148.481
C04706=1189.178,320.498,-72.121,-176.484,7.807,148.481
C04707=1189.174,320.745,-72.153,-176.482,7.810,148.481
C04708=1189.170,320.994,-72.184,-176.479,7.813,148.481
C04709=1189.166,321.241,-72.215,-176.477,7.817,148.481
C04710=1189.160,321.489,-72.247,-176.474,7.820,148.481
C04711=1189.156,321.737,-72.278,-176.472,7.822,148.481
C04712=1189.152,321.985,-72.309,-176.470,7.825,148.481
C04713=1189.148,322.233,-72.341,-176.467,7.828,148.481
C04714=1189.144,322.481,-72.372,-176.465,7.831,148.482
C04715=1189.140,322.729,-72.404,-176.462,7.834,148.482
C04716=1189.135,322.977,-72.434,-176.460,7.838,148.482
C04717=1189.132,323.225,-72.466,-176.458,7.840,148.482
C04718=1189.127,323.474,-72.497,-176.455,7.843,148.482
C04719=1189.123,323.721,-72.529,-176.453,7.846,148.482
C04720=1189.119,323.969,-72.561,-176.450,7.849,148.482
C04721=1189.115,324.217,-72.592,-176.448,7.853,148.482
C04722=1189.111,324.465,-72.623,-176.445,7.856,148.482
C04723=1189.107,324.713,-72.655,-176.443,7.859,148.482
C04724=1189.102,324.962,-72.687,-176.441,7.861,148.482
C04725=1189.098,325.209,-72.718,-176.438,7.864,148.483
C04726=1189.094,325.457,-72.750,-176.436,7.868,148.483
C04727=1189.089,325.705,-72.781,-176.433,7.871,148.483
C04728=1189.086,325.953,-72.813,-176.431,7.874,148.483
C04729=1189.082,326.201,-72.844,-176.428,7.877,148.483
C04730=1189.077,326.449,-72.876,-176.426,7.880,148.483
C04731=1189.073,326.697,-72.908,-176.424,7.883,148.483
C04732=1189.069,326.945,-72.939,-176.421,7.886,148.483
C04733=1189.065,327.193,-72.971,-176.419,7.889,148.483
C04734=1189.061,327.441,-73.003,-176.416,7.892,148.483
C04735=1189.056,327.689,-73.034,-176.414,7.895,148.483
C04736=1189.052,327.937,-73.066,-176.411,7.898,148.483
C04737=1189.048,328.184,-73.097,-176.409,7.902,148.484
C04738=1189.044,328.432,-73.129,-176.407,7.904,148.484
C04739=1189.040,328.681,-73.162,-176.405,7.907,148.484
C04740=1189.035,328.928,-73.193,-176.403,7.910,148.484
C04741=1189.031,329.177,-73.224,-176.400,7.914,148.484
C04742=1189.027,329.424,-73.256,-176.398,7.917,148.484
C04743=1189.023,329.672,-73.288,-176.395,7.920,148.484
C04744=1189.019,329.920,-73.320,-176.393,7.923,148.484
C04745=1189.015,330.168,-73.352,-176.390,7.926,148.484
C04746=1189.010,330.416,-73.384,-176.388,7.929,148.485
C04747=1189.007,330.664,-73.416,-176.386,7.932,148.485
C04748=1189.002,330.911,-73.447,-176.383,7.935,148.485
C04749=1188.998,331.160,-73.480,-176.381,7.938,148.485
C04750=1188.994,331.408,-73.512,-176.378,7.941,148.485
C04751=1188.990,331.655,-73.543,-176.376,7.945,148.485
C04752=1188.985,331.904,-73.576,-176.374,7.948,148.486
C04753=1188.982,332.152,-73.607,-176.372,7.950,148.485
C04754=1188.977,332.399,-73.639,-176.369,7.953,148.486
C04755=1188.973,332.647,-73.671,-176.367,7.957,148.486
C04756=1188.969,332.895,-73.703,-176.365,7.960,148.486
C04757=1188.964,333.143,-73.735,-176.362,7.963,148.486
C04758=1188.960,333.391,-73.767,-176.360,7.966,148.486
C04759=1188.956,333.639,-73.800,-176.357,7.969,148.486
C04760=1188.953,333.887,-73.832,-176.355,7.973,148.487
C04761=1188.948,334.134,-73.864,-176.353,7.976,148.487
C04762=1188.944,334.382,-73.896,-176.351,7.978,148.487
C04763=1188.940,334.630,-73.928,-176.348,7.982,148.487
C04764=1188.936,334.879,-73.960,-176.346,7.985,148.487
C04765=1188.931,335.126,-73.992,-176.343,7.988,148.487
C04766=1188.927,335.374,-74.025,-176.341,7.991,148.487
C04767=1188.924,335.622,-74.057,-176.339,7.995,148.488
C04768=1188.919,335.870,-74.089,-176.337,7.998,148.488
C04769=1188.915,336.118,-74.121,-176.334,8.001,148.488
C04770=1188.911,336.365,-74.154,-176.332,8.003,148.488
C04771=1188.907,336.613,-74.186,-176.330,8.007,148.488
C04772=1188.902,336.862,-74.218,-176.327,8.010,148.488
C04773=1188.898,337.109,-74.250,-176.325,8.013,148.488
C04774=1188.894,337.357,-74.283,-176.323,8.016,148.489
C04775=1188.890,337.605,-74.315,-176.321,8.020,148.489
C04776=1188.886,337.853,-74.347,-176.318,8.023,148.489
C04777=1188.882,338.101,-74.380,-176.316,8.026,148.489
C04778=1188.877,338.348,-74.412,-176.313,8.029,148.489
C04779=1188.873,338.597,-74.444,-176.312,8.032,148.489
C04780=1188.870,338.844,-74.477,-176.310,8.035,148.490
C04781=1188.865,339.092,-74.509,-176.307,8.038,148.490
C04782=1188.862,339.340,-74.542,-176.305,8.042,148.490
C04783=1188.857,339.588,-74.574,-176.302,8.045,148.490
C04784=1188.852,339.836,-74.606,-176.300,8.048,148.490
C04785=1188.848,340.114,-74.643,-176.298,8.052,148.490
C04786=1188.843,340.393,-74.679,-176.295,8.056,148.491
C04787=1188.839,340.671,-74.716,-176.292,8.059,148.491
C04788=1188.834,340.950,-74.753,-176.290,8.062,148.491
C04789=1188.830,341.198,-74.785,-176.288,8.065,148.491
C04790=1188.826,341.446,-74.818,-176.286,8.069,148.491
C04791=1188.821,341.694,-74.850,-176.283,8.072,148.492
C04792=1188.818,341.942,-74.883,-176.281,8.075,148.492
C04793=1188.814,342.190,-74.915,-176.279,8.079,148.492
C04794=1188.809,342.438,-74.949,-176.277,8.082,148.492
C04795=1188.806,342.686,-74.980,-176.274,8.085,148.492
C04796=1188.801,342.933,-75.013,-176.272,8.087,148.492
C04797=1188.797,343.181,-75.046,-176.270,8.091,148.493
C04798=1188.792,343.429,-75.079,-176.268,8.094,148.493
C04799=1188.789,343.677,-75.111,-176.265,8.097,148.493
C04800=1188.785,343.925,-75.144,-176.263,8.101,148.493
C04801=1188.780,344.173,-75.177,-176.261,8.104,148.494
C04802=1188.776,344.420,-75.210,-176.259,8.107,148.494
C04803=1188.772,344.669,-75.243,-176.256,8.111,148.494
C04804=1188.768,344.916,-75.275,-176.254,8.114,148.494
C04805=1188.764,345.164,-75.308,-176.252,8.117,148.494
C04806=1188.760,345.412,-75.342,-176.250,8.120,148.495
C04807=1188.755,345.659,-75.374,-176.248,8.123,148.495
C04808=1188.751,345.907,-75.407,-176.246,8.126,148.495
C04809=1188.748,346.154,-75.439,-176.244,8.130,148.495
C04810=1188.743,346.402,-75.472,-176.241,8.133,148.495
C04811=1188.739,346.650,-75.505,-176.239,8.136,148.496
C04812=1188.735,346.898,-75.538,-176.237,8.140,148.496
C04813=1188.731,347.146,-75.571,-176.235,8.143,148.496
C04814=1188.727,347.394,-75.604,-176.232,8.146,148.496
C04815=1188.722,347.641,-75.638,-176.230,8.150,148.497
C04816=1188.718,347.890,-75.670,-176.228,8.152,148.497
C04817=1188.715,348.137,-75.703,-176.226,8.156,148.497
C04818=1188.710,348.385,-75.736,-176.224,8.159,148.497
C04819=1188.706,348.633,-75.769,-176.222,8.162,148.497
C04820=1188.702,348.880,-75.802,-176.220,8.166,148.498
C04821=1188.698,349.128,-75.835,-176.218,8.169,148.498
C04822=1188.694,349.376,-75.868,-176.215,8.172,148.498
C04823=1188.690,349.623,-75.901,-176.213,8.176,148.499
C04824=1188.686,349.871,-75.935,-176.211,8.179,148.499
C04825=1188.681,350.119,-75.968,-176.209,8.182,148.499
C04826=1188.677,350.367,-76.000,-176.207,8.185,148.499
C04827=1188.673,350.615,-76.033,-176.205,8.189,148.500
C04828=1188.669,350.863,-76.067,-176.203,8.192,148.500
C04829=1188.665,351.110,-76.100,-176.201,8.195,148.500
C04830=1188.660,351.358,-76.133,-176.198,8.199,148.500
C04831=1188.657,351.606,-76.167,-176.196,8.202,148.500
C04832=1188.653,351.854,-76.200,-176.194,8.205,148.501
C04833=1188.649,352.101,-76.233,-176.192,8.209,148.501
C04834=1188.645,352.349,-76.267,-176.190,8.212,148.501
C04835=1188.641,352.597,-76.300,-176.188,8.215,148.502
C04836=1188.637,352.845,-76.333,-176.185,8.219,148.502
C04837=1188.632,353.092,-76.366,-176.184,8.222,148.502
C04838=1188.628,353.340,-76.399,-176.182,8.225,148.502
C04839=1188.624,353.588,-76.432,-176.180,8.228,148.503
C04840=1188.620,353.836,-76.465,-176.177,8.232,148.503
C04841=1188.616,354.083,-76.499,-176.176,8.235,148.503
C04842=1188.613,354.331,-76.533,-176.173,8.239,148.503
C04843=1188.609,354.579,-76.566,-176.171,8.242,148.504
C04844=1188.604,354.827,-76.600,-176.169,8.245,148.504
C04845=1188.599,355.075,-76.633,-176.167,8.249,148.504
C04846=1188.595,355.322,-76.666,-176.165,8.252,148.505
C04847=1188.592,355.569,-76.700,-176.163,8.256,148.505
C04848=1188.587,355.817,-76.733,-176.161,8.258,148.505
C04849=1188.583,356.065,-76.766,-176.159,8.262,148.505
C04850=1188.580,356.313,-76.800,-176.157,8.265,148.506
C04851=1188.576,356.560,-76.834,-176.155,8.268,148.506
C04852=1188.571,356.809,-76.867,-176.153,8.272,148.507
C04853=1188.567,357.056,-76.901,-176.151,8.275,148.507
C04854=1188.563,357.303,-76.934,-176.149,8.279,148.507
C04855=1188.559,357.551,-76.968,-176.147,8.282,148.507
C04856=1188.555,357.800,-77.001,-176.145,8.286,148.508
C04857=1188.551,358.047,-77.036,-176.143,8.289,148.508
C04858=1188.547,358.295,-77.069,-176.141,8.293,148.508
C04859=1188.543,358.542,-77.102,-176.139,8.295,148.509
C04860=1188.539,358.789,-77.136,-176.137,8.299,148.509
C04861=1188.535,359.038,-77.169,-176.135,8.302,148.509
C04862=1188.531,359.285,-77.204,-176.133,8.306,148.510
C04863=1188.526,359.533,-77.237,-176.131,8.309,148.510
C04864=1188.522,359.781,-77.270,-176.129,8.313,148.510
C04865=1188.518,360.028,-77.304,-176.127,8.316,148.511
C04866=1188.514,360.277,-77.338,-176.125,8.320,148.511
C04867=1188.510,360.524,-77.372,-176.124,8.322,148.511
C04868=1188.506,360.771,-77.405,-176.122,8.326,148.512
C04869=1188.502,361.019,-77.439,-176.120,8.329,148.512
C04870=1188.498,361.267,-77.473,-176.118,8.333,148.512
C04871=1188.494,361.514,-77.507,-176.116,8.337,148.513
C04872=1188.490,361.762,-77.540,-176.114,8.340,148.513
C04873=1188.486,362.010,-77.575,-176.113,8.343,148.513
C04874=1188.482,362.257,-77.609,-176.111,8.346,148.514
C04875=1188.478,362.505,-77.642,-176.109,8.350,148.514
C04876=1188.474,362.753,-77.676,-176.107,8.353,148.514
C04877=1188.469,363.000,-77.710,-176.105,8.357,148.515
C04878=1188.466,363.248,-77.744,-176.104,8.360,148.515
C04879=1188.462,363.496,-77.778,-176.101,8.363,148.516
C04880=1188.458,363.743,-77.811,-176.100,8.367,148.516
C04881=1188.454,363.991,-77.846,-176.098,8.370,148.516
C04882=1188.449,364.239,-77.879,-176.096,8.374,148.517
C04883=1188.446,364.486,-77.913,-176.095,8.377,148.517
C04884=1188.442,364.734,-77.948,-176.093,8.380,148.518
C04885=1188.438,364.982,-77.981,-176.091,8.384,148.518
C04886=1188.434,365.229,-78.015,-176.089,8.387,148.518
C04887=1188.430,365.477,-78.050,-176.088,8.390,148.519
C04888=1188.426,365.724,-78.084,-176.086,8.394,148.519
C04889=1188.421,366.006,-78.122,-176.084,8.397,148.520
C04890=1188.416,366.287,-78.161,-176.082,8.401,148.520
C04891=1188.412,366.569,-78.200,-176.080,8.405,148.520
C04892=1188.407,366.849,-78.238,-176.078,8.409,148.521
C04893=1188.403,367.097,-78.273,-176.076,8.413,148.521
C04894=1188.399,367.345,-78.306,-176.075,8.416,148.522
C04895=1188.395,367.592,-78.340,-176.073,8.419,148.522
C04896=1188.391,367.840,-78.375,-176.071,8.423,148.523
C04897=1188.387,368.087,-78.409,-176.070,8.426,148.523
C04898=1188.383,368.335,-78.443,-176.069,8.430,148.524
C04899=1188.379,368.583,-78.478,-176.067,8.433,148.524
C04900=1188.375,368.831,-78.511,-176.066,8.436,148.524
C04901=1188.371,369.079,-78.546,-176.064,8.440,148.525
C04902=1188.367,369.326,-78.580,-176.062,8.443,148.525
C04903=1188.362,369.573,-78.615,-176.061,8.446,148.526
C04904=1188.359,369.821,-78.649,-176.059,8.450,148.526
C04905=1188.354,370.069,-78.683,-176.058,8.452,148.527
C04906=1188.351,370.316,-78.717,-176.057,8.456,148.527
C04907=1188.347,370.564,-78.752,-176.055,8.460,148.528
C04908=1188.343,370.811,-78.786,-176.054,8.463,148.528
C04909=1188.339,371.059,-78.821,-176.052,8.466,148.528
C04910=1188.334,371.306,-78.855,-176.051,8.469,148.529
C04911=1188.331,371.554,-78.889,-176.049,8.473,148.529
C04912=1188.327,371.802,-78.924,-176.048,8.476,148.530
C04913=1188.323,372.049,-78.958,-176.046,8.480,148.530
C04914=1188.319,372.297,-78.993,-176.045,8.483,148.531
C04915=1188.314,372.544,-79.027,-176.043,8.486,148.531
C04916=1188.311,372.792,-79.061,-176.042,8.489,148.532
C04917=1188.306,373.040,-79.096,-176.041,8.493,148.532
C04918=1188.302,373.288,-79.131,-176.040,8.496,148.533
C04919=1188.299,373.535,-79.164,-176.038,8.499,148.533
C04920=1188.294,373.782,-79.199,-176.037,8.502,148.534
C04921=1188.291,374.030,-79.233,-176.035,8.506,148.534
C04922=1188.286,374.277,-79.268,-176.034,8.509,148.535
C04923=1188.282,374.526,-79.302,-176.033,8.513,148.535
C04924=1188.278,374.773,-79.336,-176.031,8.516,148.536
C04925=1188.274,375.021,-79.371,-176.030,8.520,148.536
C04926=1188.270,375.268,-79.406,-176.029,8.522,148.537
C04927=1188.267,375.515,-79.441,-176.028,8.525,148.537
C04928=1188.262,375.763,-79.475,-176.026,8.529,148.538
C04929=1188.258,376.011,-79.510,-176.025,8.532,148.538
C04930=1188.254,376.258,-79.544,-176.024,8.536,148.539
C04931=1188.251,376.506,-79.579,-176.023,8.539,148.539
C04932=1188.246,376.753,-79.614,-176.022,8.542,148.540
C04933=1188.242,377.001,-79.649,-176.020,8.546,148.540
C04934=1188.238,377.248,-79.683,-176.019,8.549,148.541
C04935=1188.235,377.496,-79.717,-176.018,8.552,148.541
C04936=1188.230,377.744,-79.752,-176.017,8.555,148.542
C04937=1188.226,377.991,-79.787,-176.016,8.558,148.542
C04938=1188.222,378.239,-79.822,-176.015,8.561,148.543
C04939=1188.219,378.486,-79.856,-176.014,8.564,148.543
C04940=1188.214,378.734,-79.891,-176.012,8.568,148.544
C04941=1188.210,378.981,-79.926,-176.011,8.571,148.544
C04942=1188.206,379.229,-79.961,-176.011,8.574,148.545
C04943=1188.202,379.477,-79.995,-176.009,8.577,148.545
C04944=1188.198,379.723,-80.030,-176.008,8.580,148.546
C04945=1188.194,379.972,-80.065,-176.007,8.584,148.547
C04946=1188.190,380.219,-80.099,-176.006,8.587,148.547
C04947=1188.186,380.467,-80.134,-176.005,8.590,148.548
C04948=1188.181,380.714,-80.169,-176.004,8.593,148.548
C04949=1188.178,380.962,-80.203,-176.003,8.596,148.549
C04950=1188.174,381.208,-80.239,-176.003,8.599,148.549
C04951=1188.170,381.457,-80.274,-176.001,8.603,148.550
C04952=1188.166,381.705,-80.308,-176.000,8.606,148.550
C04953=1188.162,381.951,-80.344,-175.999,8.609,148.551
C04954=1188.158,382.200,-80.378,-175.998,8.612,148.552
C04955=1188.154,382.447,-80.412,-175.998,8.615,148.552
C04956=1188.150,382.694,-80.448,-175.997,8.618,148.553
C04957=1188.146,382.942,-80.482,-175.996,8.621,148.553
C04958=1188.142,383.189,-80.518,-175.995,8.625,148.554
C04959=1188.138,383.437,-80.553,-175.994,8.628,148.554
C04960=1188.134,383.684,-80.588,-175.994,8.631,148.555
C04961=1188.130,383.932,-80.623,-175.993,8.634,148.556
C04962=1188.125,384.180,-80.657,-175.992,8.637,148.556
C04963=1188.122,384.427,-80.692,-175.991,8.640,148.557
C04964=1188.118,384.675,-80.727,-175.990,8.643,148.557
C04965=1188.114,384.922,-80.762,-175.989,8.646,148.558
C04966=1188.110,385.170,-80.797,-175.988,8.649,148.558
C04967=1188.106,385.417,-80.832,-175.989,8.652,148.559
C04968=1188.102,385.665,-80.867,-175.988,8.655,148.560
C04969=1188.098,385.912,-80.902,-175.987,8.658,148.560
C04970=1188.094,386.160,-80.937,-175.986,8.661,148.561
C04971=1188.090,386.407,-80.972,-175.985,8.664,148.561
C04972=1188.085,386.655,-81.007,-175.984,8.667,148.562
C04973=1188.082,386.902,-81.042,-175.984,8.669,148.562
C04974=1188.078,387.150,-81.078,-175.983,8.672,148.563
C04975=1188.074,387.397,-81.113,-175.983,8.676,148.564
C04976=1188.071,387.644,-81.147,-175.982,8.679,148.564
C04977=1188.067,387.892,-81.182,-175.982,8.681,148.565
C04978=1188.062,388.139,-81.217,-175.981,8.684,148.565
C04979=1188.058,388.387,-81.252,-175.980,8.687,148.566
C04980=1188.054,388.634,-81.287,-175.980,8.690,148.567
C04981=1188.051,388.882,-81.323,-175.979,8.693,148.567
C04982=1188.047,389.130,-81.358,-175.979,8.696,148.568
C04983=1188.042,389.376,-81.393,-175.978,8.698,148.568
C04984=1188.038,389.625,-81.428,-175.977,8.701,148.569
C04985=1188.035,389.872,-81.463,-175.977,8.705,148.570
C04986=1188.030,390.119,-81.499,-175.977,8.707,148.570
C04987=1188.026,390.367,-81.533,-175.976,8.710,148.571
C04988=1188.023,390.615,-81.569,-175.976,8.712,148.571
C04989=1188.018,390.861,-81.604,-175.975,8.715,148.572
C04990=1188.015,391.109,-81.639,-175.975,8.718,148.573
C04991=1188.011,391.357,-81.675,-175.974,8.721,148.573
C04992=1188.007,391.604,-81.710,-175.974,8.723,148.574
C04993=1188.002,391.888,-81.750,-175.974,8.727,148.575
C04994=1187.997,392.171,-81.791,-175.973,8.730,148.575
C04995=1187.993,392.455,-81.831,-175.973,8.733,148.576
C04996=1187.988,392.738,-81.871,-175.972,8.736,148.577
C04997=1187.984,392.987,-81.906,-175.972,8.739,148.577
C04998=1187.981,393.234,-81.942,-175.971,8.742,148.578
C04999=1187.976,393.481,-81.977,-175.971,8.744,148.578
C05000=1187.973,393.728,-82.013,-175.970,8.747,148.579
C05001=1187.969,393.977,-82.047,-175.970,8.750,148.580
C05002=1187.965,394.223,-82.083,-175.970,8.752,148.580
C05003=1187.961,394.471,-82.118,-175.969,8.755,148.581
C05004=1187.957,394.718,-82.154,-175.969,8.758,148.581
C05005=1187.952,394.966,-82.189,-175.969,8.760,148.582
C05006=1187.948,395.214,-82.224,-175.968,8.763,148.583
C05007=1187.945,395.461,-82.260,-175.968,8.765,148.583
C05008=1187.940,395.708,-82.295,-175.968,8.768,148.584
C05009=1187.936,395.956,-82.330,-175.968,8.771,148.584
C05010=1187.933,396.203,-82.365,-175.967,8.773,148.585
C05011=1187.929,396.451,-82.401,-175.967,8.776,148.586
C05012=1187.925,396.698,-82.436,-175.967,8.778,148.586
C05013=1187.921,396.945,-82.472,-175.966,8.781,148.587
C05014=1187.917,397.193,-82.506,-175.966,8.784,148.587
C05015=1187.912,397.441,-82.542,-175.966,8.786,148.588
C05016=1187.908,397.688,-82.578,-175.966,8.788,148.589
C05017=1187.905,397.936,-82.613,-175.966,8.791,148.589
C05018=1187.901,398.183,-82.649,-175.965,8.794,148.590
C05019=1187.897,398.430,-82.683,-175.965,8.796,148.590
C05020=1187.893,398.678,-82.719,-175.965,8.799,148.591
C05021=1187.889,398.925,-82.754,-175.965,8.801,148.591
C05022=1187.885,399.172,-82.790,-175.965,8.803,148.592
C05023=1187.881,399.420,-82.826,-175.965,8.806,148.593
C05024=1187.877,399.668,-82.861,-175.964,8.809,148.593
C05025=1187.873,399.915,-82.897,-175.964,8.811,148.594
C05026=1187.869,400.162,-82.931,-175.964,8.814,148.595
C05027=1187.865,400.410,-82.967,-175.964,8.816,148.595
C05028=1187.861,400.657,-83.002,-175.963,8.818,148.596
C05029=1187.858,400.905,-83.038,-175.963,8.821,148.596
C05030=1187.853,401.152,-83.074,-175.963,8.823,148.597
C05031=1187.849,401.400,-83.109,-175.963,8.825,148.597
C05032=1187.845,401.647,-83.145,-175.963,8.828,148.598
C05033=1187.842,401.895,-83.180,-175.963,8.830,148.599
C05034=1187.837,402.141,-83.216,-175.963,8.832,148.599
C05035=1187.833,402.389,-83.250,-175.962,8.835,148.600
C05036=1187.829,402.637,-83.287,-175.963,8.837,148.600
C05037=1187.825,402.885,-83.322,-175.962,8.839,148.601
C05038=1187.821,403.132,-83.357,-175.962,8.842,148.601
C05039=1187.817,403.379,-83.393,-175.962,8.844,148.602
C05040=1187.814,403.627,-83.428,-175.962,8.847,148.603
C05041=1187.809,403.874,-83.465,-175.962,8.849,148.603
C05042=1187.805,404.121,-83.500,-175.962,8.851,148.604
C05043=1187.801,404.369,-83.535,-175.961,8.853,148.604
C05044=1187.798,404.616,-83.571,-175.961,8.856,148.605
C05045=1187.794,404.864,-83.606,-175.961,8.858,148.606
C05046=1187.790,405.112,-83.643,-175.961,8.860,148.606
C05047=1187.785,405.358,-83.678,-175.961,8.863,148.607
C05048=1187.782,405.606,-83.713,-175.961,8.865,148.607
C05049=1187.778,405.853,-83.749,-175.961,8.867,148.608
C05050=1187.774,406.101,-83.784,-175.961,8.869,148.608
C05051=1187.769,406.348,-83.820,-175.961,8.871,148.609
C05052=1187.766,406.595,-83.856,-175.961,8.874,148.610
C05053=1187.762,406.843,-83.891,-175.961,8.876,148.610
C05054=1187.758,407.090,-83.927,-175.960,8.878,148.611
C05055=1187.754,407.338,-83.963,-175.960,8.881,148.611
C05056=1187.750,407.585,-83.998,-175.960,8.883,148.612
C05057=1187.746,407.833,-84.034,-175.961,8.885,148.612
C05058=1187.743,408.080,-84.069,-175.960,8.887,148.613
C05059=1187.739,408.328,-84.105,-175.960,8.889,148.613
C05060=1187.734,408.575,-84.141,-175.960,8.891,148.614
C05061=1187.730,408.822,-84.176,-175.960,8.894,148.614
C05062=1187.727,409.070,-84.212,-175.960,8.895,148.615
C05063=1187.723,409.317,-84.247,-175.960,8.898,148.616
C05064=1187.718,409.565,-84.283,-175.960,8.900,148.616
C05065=1187.715,409.812,-84.319,-175.960,8.902,148.617
C05066=1187.711,410.059,-84.354,-175.959,8.904,148.617
C05067=1187.707,410.307,-84.390,-175.960,8.906,148.618
C05068=1187.702,410.555,-84.426,-175.959,8.908,148.618
C05069=1187.699,410.802,-84.461,-175.960,8.911,148.619
C05070=1187.695,411.050,-84.497,-175.959,8.913,148.619
C05071=1187.690,411.297,-84.533,-175.960,8.914,148.620
C05072=1187.686,411.544,-84.568,-175.959,8.917,148.620
C05073=1187.683,411.791,-84.604,-175.959,8.919,148.621
C05074=1187.679,412.039,-84.640,-175.959,8.920,148.621
C05075=1187.675,412.286,-84.676,-175.959,8.923,148.622
C05076=1187.671,412.534,-84.712,-175.959,8.925,148.622
C05077=1187.667,412.781,-84.747,-175.959,8.927,148.623
C05078=1187.663,413.028,-84.783,-175.959,8.929,148.624
C05079=1187.659,413.276,-84.818,-175.959,8.931,148.624
C05080=1187.655,413.523,-84.854,-175.959,8.933,148.625
C05081=1187.652,413.771,-84.890,-175.959,8.935,148.625
C05082=1187.647,414.018,-84.925,-175.959,8.937,148.626
C05083=1187.643,414.265,-84.962,-175.959,8.939,148.626
C05084=1187.640,414.512,-84.997,-175.959,8.941,148.627
C05085=1187.635,414.760,-85.033,-175.959,8.943,148.627
C05086=1187.632,415.008,-85.069,-175.958,8.945,148.628
C05087=1187.628,415.255,-85.104,-175.959,8.947,148.628
C05088=1187.623,415.502,-85.140,-175.959,8.949,148.629
C05089=1187.618,415.908,-85.199,-175.959,8.953,148.630
C05090=1187.614,416.314,-85.258,-175.959,8.955,148.630
C05091=1187.613,416.719,-85.316,-175.958,8.959,148.631
C05092=1187.616,417.123,-85.373,-175.959,8.961,148.632
C05093=1187.195,417.125,-85.414,-175.962,8.972,148.635
C05094=1187.191,416.717,-85.356,-175.961,8.969,148.635
C05095=1187.192,416.309,-85.298,-175.962,8.966,148.634
C05096=1187.196,415.900,-85.239,-175.962,8.963,148.633
C05097=1187.203,415.492,-85.180,-175.962,8.960,148.632
C05098=1187.206,415.244,-85.144,-175.962,8.957,148.632
C05099=1187.210,414.997,-85.108,-175.962,8.956,148.631
C05100=1187.214,414.749,-85.072,-175.962,8.954,148.631
C05101=1187.218,414.502,-85.037,-175.962,8.952,148.630
C05102=1187.222,414.254,-85.000,-175.962,8.950,148.630
C05103=1187.226,414.007,-84.965,-175.962,8.948,148.629
C05104=1187.230,413.760,-84.930,-175.962,8.946,148.629
C05105=1187.234,413.512,-84.894,-175.962,8.944,148.628
C05106=1187.238,413.265,-84.857,-175.962,8.942,148.628
C05107=1187.241,413.018,-84.822,-175.962,8.940,148.627
C05108=1187.245,412.770,-84.786,-175.962,8.938,148.627
C05109=1187.250,412.523,-84.750,-175.962,8.936,148.626
C05110=1187.254,412.275,-84.715,-175.962,8.933,148.625
C05111=1187.257,412.028,-84.679,-175.962,8.932,148.625
C05112=1187.262,411.780,-84.643,-175.962,8.930,148.624
C05113=1187.265,411.533,-84.608,-175.962,8.927,148.624
C05114=1187.270,411.286,-84.572,-175.963,8.925,148.623
C05115=1187.273,411.038,-84.537,-175.962,8.924,148.623
C05116=1187.278,410.790,-84.501,-175.963,8.921,148.622
C05117=1187.281,410.544,-84.464,-175.962,8.919,148.622
C05118=1187.285,410.296,-84.429,-175.963,8.917,148.621
C05119=1187.288,410.049,-84.393,-175.962,8.915,148.621
C05120=1187.294,409.801,-84.358,-175.963,8.913,148.620
C05121=1187.297,409.554,-84.322,-175.963,8.911,148.620
C05122=1187.301,409.306,-84.286,-175.963,8.908,148.619
C05123=1187.305,409.059,-84.250,-175.962,8.907,148.619
C05124=1187.309,408.811,-84.215,-175.963,8.904,148.618
C05125=1187.313,408.564,-84.180,-175.963,8.902,148.617
C05126=1187.317,408.317,-84.144,-175.963,8.900,148.617
C05127=1187.321,408.069,-84.108,-175.963,8.898,148.616
C05128=1187.325,407.822,-84.072,-175.963,8.896,148.616
C05129=1187.329,407.574,-84.037,-175.963,8.894,148.615
C05130=1187.333,407.327,-84.002,-175.963,8.891,148.615
C05131=1187.336,407.080,-83.966,-175.963,8.889,148.614
C05132=1187.341,406.832,-83.930,-175.964,8.887,148.614
C05133=1187.345,406.584,-83.894,-175.964,8.884,148.613
C05134=1187.348,406.337,-83.859,-175.963,8.883,148.612
C05135=1187.352,406.090,-83.824,-175.963,8.880,148.612
C05136=1187.357,405.842,-83.788,-175.964,8.878,148.611
C05137=1187.361,405.595,-83.752,-175.964,8.876,148.611
C05138=1187.364,405.347,-83.716,-175.964,8.873,148.610
C05139=1187.368,405.101,-83.681,-175.964,8.871,148.610
C05140=1187.372,404.853,-83.646,-175.964,8.869,148.609
C05141=1187.377,404.605,-83.610,-175.964,8.866,148.608
C05142=1187.380,404.358,-83.574,-175.964,8.864,148.608
C05143=1187.384,404.110,-83.538,-175.965,8.862,148.607
C05144=1187.388,403.863,-83.503,-175.964,8.860,148.607
C05145=1187.392,403.616,-83.468,-175.964,8.858,148.606
C05146=1187.396,403.368,-83.432,-175.964,8.855,148.606
C05147=1187.400,403.121,-83.396,-175.965,8.853,148.605
C05148=1187.404,402.874,-83.361,-175.965,8.851,148.605
C05149=1187.408,402.626,-83.325,-175.965,8.848,148.604
C05150=1187.411,402.379,-83.290,-175.965,8.846,148.603
C05151=1187.416,402.131,-83.254,-175.965,8.844,148.603
C05152=1187.420,401.884,-83.219,-175.965,8.841,148.602
C05153=1187.424,401.636,-83.184,-175.965,8.839,148.602
C05154=1187.428,401.389,-83.148,-175.966,8.837,148.601
C05155=1187.431,401.141,-83.113,-175.966,8.834,148.601
C05156=1187.436,400.894,-83.077,-175.966,8.831,148.600
C05157=1187.440,400.646,-83.041,-175.966,8.829,148.599
C05158=1187.444,400.399,-83.006,-175.967,8.827,148.599
C05159=1187.447,400.151,-82.970,-175.966,8.824,148.598
C05160=1187.452,399.905,-82.935,-175.967,8.822,148.597
C05161=1187.455,399.657,-82.899,-175.967,8.819,148.597
C05162=1187.459,399.409,-82.865,-175.967,8.817,148.596
C05163=1187.464,399.161,-82.828,-175.967,8.815,148.596
C05164=1187.468,398.914,-82.793,-175.967,8.812,148.595
C05165=1187.472,398.667,-82.758,-175.967,8.810,148.594
C05166=1187.475,398.419,-82.722,-175.968,8.807,148.594
C05167=1187.479,398.172,-82.687,-175.968,8.804,148.593
C05168=1187.483,397.925,-82.651,-175.968,8.802,148.593
C05169=1187.487,397.677,-82.617,-175.968,8.800,148.592
C05170=1187.492,397.429,-82.580,-175.968,8.797,148.592
C05171=1187.496,397.182,-82.545,-175.969,8.794,148.591
C05172=1187.499,396.935,-82.510,-175.969,8.792,148.590
C05173=1187.503,396.687,-82.474,-175.969,8.789,148.590
C05174=1187.507,396.439,-82.439,-175.970,8.787,148.589
C05175=1187.511,396.193,-82.404,-175.970,8.784,148.588
C05176=1187.515,395.945,-82.369,-175.970,8.781,148.588
C05177=1187.519,395.698,-82.333,-175.970,8.779,148.587
C05178=1187.523,395.451,-82.298,-175.971,8.777,148.587
C05179=1187.527,395.203,-82.263,-175.971,8.774,148.586
C05180=1187.531,394.955,-82.227,-175.971,8.771,148.586
C05181=1187.535,394.707,-82.191,-175.972,8.769,148.585
C05182=1187.539,394.460,-82.156,-175.972,8.766,148.584
C05183=1187.543,394.212,-82.121,-175.972,8.763,148.584
C05184=1187.547,393.965,-82.086,-175.972,8.761,148.583
C05185=1187.551,393.718,-82.051,-175.973,8.758,148.582
C05186=1187.555,393.471,-82.015,-175.973,8.755,148.582
C05187=1187.559,393.222,-81.980,-175.974,8.752,148.581
C05188=1187.563,392.976,-81.945,-175.974,8.750,148.581
C05189=1187.567,392.728,-81.909,-175.974,8.747,148.580
C05190=1187.571,392.444,-81.869,-175.975,8.744,148.579
C05191=1187.576,392.161,-81.829,-175.975,8.741,148.579
C05192=1187.581,391.877,-81.789,-175.976,8.738,148.578
C05193=1187.585,391.593,-81.748,-175.976,8.735,148.577
C05194=1187.589,391.346,-81.712,-175.977,8.732,148.577
C05195=1187.593,391.098,-81.678,-175.977,8.729,148.576
C05196=1187.597,390.851,-81.642,-175.977,8.727,148.575
C05197=1187.601,390.603,-81.607,-175.978,8.723,148.575
C05198=1187.605,390.356,-81.572,-175.979,8.720,148.574
C05199=1187.609,390.109,-81.537,-175.979,8.718,148.574
C05200=1187.612,389.861,-81.501,-175.979,8.715,148.573
C05201=1187.617,389.614,-81.467,-175.980,8.712,148.572
C05202=1187.621,389.366,-81.431,-175.980,8.709,148.572
C05203=1187.624,389.119,-81.396,-175.981,8.706,148.571
C05204=1187.629,388.871,-81.361,-175.981,8.704,148.571
C05205=1187.633,388.624,-81.326,-175.982,8.701,148.570
C05206=1187.637,388.376,-81.291,-175.983,8.697,148.569
C05207=1187.641,388.129,-81.256,-175.983,8.695,148.569
C05208=1187.644,387.881,-81.220,-175.984,8.692,148.568
C05209=1187.648,387.633,-81.185,-175.985,8.689,148.568
C05210=1187.653,387.386,-81.150,-175.985,8.687,148.567
C05211=1187.657,387.138,-81.115,-175.986,8.684,148.567
C05212=1187.661,386.891,-81.080,-175.986,8.681,148.566
C05213=1187.665,386.643,-81.045,-175.987,8.677,148.565
C05214=1187.669,386.396,-81.010,-175.988,8.674,148.565
C05215=1187.673,386.148,-80.975,-175.988,8.672,148.564
C05216=1187.677,385.901,-80.940,-175.989,8.669,148.564
C05217=1187.680,385.654,-80.905,-175.989,8.666,148.563
C05218=1187.684,385.406,-80.870,-175.990,8.663,148.562
C05219=1187.688,385.159,-80.835,-175.991,8.659,148.562
C05220=1187.693,384.911,-80.800,-175.992,8.656,148.561
C05221=1187.696,384.664,-80.765,-175.993,8.653,148.561
C05222=1187.700,384.416,-80.730,-175.993,8.650,148.560
C05223=1187.704,384.169,-80.695,-175.994,8.647,148.559
C05224=1187.708,383.921,-80.660,-175.994,8.645,148.559
C05225=1187.713,383.673,-80.625,-175.995,8.642,148.558
C05226=1187.717,383.426,-80.590,-175.996,8.639,148.558
C05227=1187.721,383.178,-80.555,-175.997,8.635,148.557
C05228=1187.724,382.931,-80.520,-175.998,8.632,148.557
C05229=1187.728,382.683,-80.485,-175.999,8.629,148.556
C05230=1187.732,382.436,-80.450,-176.000,8.626,148.556
C05231=1187.736,382.188,-80.415,-176.001,8.623,148.555
C05232=1187.741,381.941,-80.381,-176.002,8.619,148.554
C05233=1187.745,381.693,-80.345,-176.003,8.616,148.554
C05234=1187.749,381.445,-80.311,-176.004,8.613,148.553
C05235=1187.752,381.199,-80.276,-176.004,8.610,148.553
C05236=1187.756,380.951,-80.241,-176.005,8.607,148.552
C05237=1187.761,380.703,-80.207,-176.006,8.604,148.552
C05238=1187.764,380.456,-80.171,-176.007,8.601,148.551
C05239=1187.769,380.208,-80.137,-176.009,8.597,148.550
C05240=1187.773,379.960,-80.102,-176.009,8.594,148.550
C05241=1187.776,379.714,-80.067,-176.011,8.591,148.549
C05242=1187.780,379.466,-80.032,-176.011,8.588,148.549
C05243=1187.785,379.218,-79.998,-176.012,8.585,148.548
C05244=1187.789,378.971,-79.962,-176.014,8.581,148.548
C05245=1187.793,378.723,-79.928,-176.015,8.578,148.547
C05246=1187.796,378.475,-79.894,-176.016,8.575,148.547
C05247=1187.800,378.227,-79.859,-176.016,8.572,148.546
C05248=1187.805,377.980,-79.824,-176.018,8.569,148.546
C05249=1187.809,377.732,-79.789,-176.019,8.566,148.545
C05250=1187.812,377.485,-79.755,-176.020,8.562,148.545
C05251=1187.816,377.237,-79.720,-176.022,8.559,148.544
C05252=1187.821,376.990,-79.685,-176.022,8.556,148.543
C05253=1187.825,376.742,-79.650,-176.024,8.553,148.543
C05254=1187.828,376.495,-79.616,-176.025,8.549,148.542
C05255=1187.832,376.247,-79.581,-176.026,8.546,148.542
C05256=1187.837,376.000,-79.547,-176.027,8.543,148.542
C05257=1187.841,375.752,-79.511,-176.028,8.539,148.541
C05258=1187.844,375.505,-79.478,-176.030,8.536,148.540
C05259=1187.849,375.258,-79.443,-176.031,8.532,148.540
C05260=1187.853,375.009,-79.408,-176.032,8.530,148.539
C05261=1187.857,374.762,-79.374,-176.034,8.527,148.539
C05262=1187.861,374.514,-79.340,-176.035,8.523,148.538
C05263=1187.865,374.267,-79.305,-176.036,8.520,148.538
C05264=1187.868,374.020,-79.270,-176.038,8.516,148.537
C05265=1187.873,373.772,-79.236,-176.039,8.513,148.537
C05266=1187.877,373.524,-79.201,-176.040,8.509,148.536
C05267=1187.881,373.277,-79.167,-176.041,8.507,148.536
C05268=1187.885,373.029,-79.132,-176.043,8.503,148.536
C05269=1187.889,372.781,-79.098,-176.044,8.500,148.535
C05270=1187.892,372.534,-79.063,-176.046,8.496,148.535
C05271=1187.897,372.286,-79.029,-176.047,8.494,148.534
C05272=1187.901,372.039,-78.995,-176.048,8.490,148.534
C05273=1187.905,371.791,-78.960,-176.050,8.487,148.533
C05274=1187.909,371.543,-78.926,-176.051,8.483,148.533
C05275=1187.913,371.296,-78.892,-176.053,8.480,148.532
C05276=1187.917,371.048,-78.857,-176.054,8.476,148.532
C05277=1187.920,370.800,-78.823,-176.056,8.473,148.531
C05278=1187.925,370.553,-78.788,-176.057,8.470,148.531
C05279=1187.929,370.306,-78.754,-176.059,8.466,148.530
C05280=1187.933,370.058,-78.720,-176.060,8.463,148.530
C05281=1187.937,369.810,-78.685,-176.062,8.460,148.529
C05282=1187.941,369.563,-78.651,-176.063,8.456,148.529
C05283=1187.945,369.315,-78.617,-176.065,8.453,148.529
C05284=1187.949,369.067,-78.583,-176.066,8.450,148.528
C05285=1187.953,368.819,-78.549,-176.068,8.446,148.528
C05286=1187.957,368.572,-78.515,-176.069,8.443,148.527
C05287=1187.962,368.325,-78.480,-176.071,8.440,148.527
C05288=1187.966,368.077,-78.445,-176.073,8.436,148.526
C05289=1187.969,367.830,-78.411,-176.074,8.433,148.526
C05290=1187.974,367.582,-78.377,-176.076,8.429,148.525
C05291=1187.978,367.334,-78.343,-176.077,8.426,148.525
C05292=1187.982,367.086,-78.309,-176.079,8.423,148.525
C05293=1187.985,366.838,-78.275,-176.080,8.419,148.524
C05294=1187.990,366.558,-78.236,-176.082,8.416,148.524
C05295=1187.994,366.277,-78.197,-176.084,8.412,148.523
C05296=1188.000,365.995,-78.159,-176.086,8.407,148.523
C05297=1188.004,365.714,-78.120,-176.088,8.404,148.522
C05298=1188.008,365.467,-78.086,-176.090,8.400,148.522
C05299=1188.012,365.218,-78.052,-176.091,8.397,148.522
C05300=1188.016,364.971,-78.018,-176.093,8.394,148.521
C05301=1188.021,364.723,-77.984,-176.095,8.390,148.521
C05302=1188.024,364.475,-77.950,-176.097,8.387,148.520
C05303=1188.028,364.228,-77.916,-176.098,8.384,148.520
C05304=1188.033,363.980,-77.882,-176.100,8.380,148.520
C05305=1188.036,363.733,-77.848,-176.102,8.377,148.519
C05306=1188.040,363.485,-77.815,-176.104,8.373,148.519
C05307=1188.045,363.237,-77.780,-176.106,8.370,148.519
C05308=1188.048,362.990,-77.746,-176.107,8.367,148.518
C05309=1188.053,362.742,-77.712,-176.109,8.363,148.518
C05310=1188.056,362.494,-77.678,-176.111,8.360,148.517
C05311=1188.060,362.247,-77.644,-176.113,8.356,148.517
C05312=1188.065,361.999,-77.610,-176.115,8.353,148.517
C05313=1188.068,361.751,-77.576,-176.116,8.350,148.516
C05314=1188.073,361.504,-77.543,-176.118,8.347,148.516
C05315=1188.076,361.257,-77.509,-176.120,8.343,148.516
C05316=1188.081,361.008,-77.475,-176.122,8.339,148.515
C05317=1188.084,360.761,-77.441,-176.124,8.336,148.515
C05318=1188.089,360.513,-77.408,-176.126,8.333,148.515
C05319=1188.093,360.266,-77.374,-176.128,8.329,148.514
C05320=1188.097,360.017,-77.340,-176.130,8.326,148.514
C05321=1188.101,359.770,-77.306,-176.131,8.323,148.514
C05322=1188.105,359.522,-77.273,-176.134,8.319,148.513
C05323=1188.109,359.275,-77.239,-176.135,8.316,148.513
C05324=1188.113,359.027,-77.206,-176.138,8.313,148.513
C05325=1188.117,358.779,-77.172,-176.140,8.309,148.512
C05326=1188.121,358.532,-77.138,-176.142,8.306,148.512
C05327=1188.126,358.284,-77.104,-176.144,8.302,148.512
C05328=1188.129,358.037,-77.071,-176.146,8.299,148.511
C05329=1188.134,357.789,-77.037,-176.148,8.295,148.511
C05330=1188.137,357.540,-77.004,-176.149,8.293,148.511
C05331=1188.141,357.293,-76.970,-176.151,8.289,148.510
C05332=1188.146,357.045,-76.936,-176.153,8.286,148.510
C05333=1188.150,356.797,-76.903,-176.156,8.282,148.510
C05334=1188.154,356.550,-76.869,-176.157,8.279,148.509
C05335=1188.157,356.302,-76.836,-176.160,8.275,148.509
C05336=1188.161,356.054,-76.803,-176.161,8.272,148.509
C05337=1188.166,355.806,-76.769,-176.164,8.268,148.508
C05338=1188.169,355.559,-76.736,-176.166,8.265,148.508
C05339=1188.174,355.311,-76.702,-176.168,8.261,148.508
C05340=1188.178,355.064,-76.669,-176.170,8.258,148.508
C05341=1188.183,354.816,-76.636,-176.172,8.255,148.507
C05342=1188.186,354.568,-76.601,-176.173,8.252,148.507
C05343=1188.190,354.320,-76.568,-176.176,8.249,148.507
C05344=1188.194,354.073,-76.535,-176.178,8.245,148.507
C05345=1188.198,353.825,-76.502,-176.180,8.242,148.506
C05346=1188.202,353.577,-76.469,-176.182,8.238,148.506
C05347=1188.207,353.329,-76.436,-176.184,8.235,148.506
C05348=1188.211,353.082,-76.402,-176.187,8.232,148.505
C05349=1188.215,352.834,-76.368,-176.188,8.228,148.505
C05350=1188.219,352.587,-76.335,-176.191,8.225,148.505
C05351=1188.224,352.339,-76.302,-176.193,8.221,148.505
C05352=1188.227,352.090,-76.268,-176.195,8.218,148.504
C05353=1188.231,351.843,-76.235,-176.197,8.215,148.504
C05354=1188.235,351.595,-76.202,-176.199,8.212,148.504
C05355=1188.239,351.347,-76.169,-176.201,8.209,148.504
C05356=1188.244,351.099,-76.135,-176.203,8.205,148.503
C05357=1188.248,350.852,-76.102,-176.205,8.202,148.503
C05358=1188.252,350.604,-76.069,-176.208,8.199,148.503
C05359=1188.256,350.356,-76.036,-176.209,8.195,148.502
C05360=1188.260,350.109,-76.003,-176.212,8.192,148.502
C05361=1188.264,349.861,-75.970,-176.214,8.188,148.502
C05362=1188.268,349.613,-75.937,-176.216,8.185,148.502
C05363=1188.272,349.366,-75.904,-176.218,8.182,148.502
C05364=1188.276,349.118,-75.871,-176.221,8.178,148.501
C05365=1188.280,348.870,-75.838,-176.222,8.176,148.501
C05366=1188.284,348.622,-75.804,-176.225,8.173,148.501
C05367=1188.288,348.375,-75.771,-176.226,8.169,148.501
C05368=1188.293,348.126,-75.739,-176.229,8.166,148.500
C05369=1188.297,347.879,-75.706,-176.231,8.162,148.500
C05370=1188.301,347.631,-75.673,-176.233,8.159,148.500
C05371=1188.305,347.383,-75.639,-176.235,8.156,148.500
C05372=1188.309,347.135,-75.606,-176.238,8.152,148.499
C05373=1188.314,346.888,-75.573,-176.240,8.149,148.499
C05374=1188.317,346.640,-75.541,-176.242,8.146,148.499
C05375=1188.321,346.392,-75.508,-176.244,8.142,148.499
C05376=1188.326,346.144,-75.475,-176.246,8.140,148.499
C05377=1188.330,345.897,-75.442,-176.248,8.137,148.498
C05378=1188.334,345.648,-75.409,-176.250,8.133,148.498
C05379=1188.338,345.400,-75.376,-176.253,8.130,148.498
C05380=1188.342,345.153,-75.344,-176.255,8.127,148.498
C05381=1188.346,344.905,-75.310,-176.257,8.123,148.497
C05382=1188.350,344.657,-75.278,-176.259,8.120,148.497
C05383=1188.355,344.410,-75.245,-176.262,8.117,148.497
C05384=1188.359,344.162,-75.212,-176.264,8.113,148.497
C05385=1188.363,343.914,-75.180,-176.266,8.110,148.497
C05386=1188.367,343.666,-75.147,-176.268,8.107,148.496
C05387=1188.371,343.419,-75.114,-176.270,8.104,148.496
C05388=1188.376,343.170,-75.081,-176.272,8.101,148.496
C05389=1188.379,342.923,-75.049,-176.275,8.098,148.496
C05390=1188.383,342.675,-75.016,-176.277,8.094,148.496
C05391=1188.387,342.427,-74.983,-176.280,8.091,148.496
C05392=1188.392,342.179,-74.950,-176.282,8.088,148.495
C05393=1188.396,341.932,-74.919,-176.284,8.085,148.495
C05394=1188.400,341.684,-74.886,-176.286,8.081,148.495
C05395=1188.405,341.436,-74.853,-176.289,8.078,148.495
C05396=1188.409,341.188,-74.820,-176.291,8.075,148.494
C05397=1188.412,340.940,-74.788,-176.293,8.072,148.494
C05398=1188.417,340.661,-74.752,-176.295,8.068,148.494
C05399=1188.422,340.382,-74.714,-176.298,8.065,148.494
C05400=1188.426,340.104,-74.678,-176.301,8.061,148.494
C05401=1188.431,339.825,-74.642,-176.303,8.058,148.494
C05402=1188.435,339.577,-74.609,-176.305,8.054,148.493
C05403=1188.439,339.329,-74.577,-176.308,8.051,148.493
C05404=1188.443,339.081,-74.544,-176.310,8.048,148.493
C05405=1188.448,338.834,-74.512,-176.313,8.045,148.493
C05406=1188.452,338.586,-74.479,-176.314,8.042,148.493
C05407=1188.456,338.338,-74.447,-176.316,8.039,148.492
C05408=1188.460,338.090,-74.415,-176.319,8.035,148.492
C05409=1188.464,337.842,-74.382,-176.321,8.032,148.492
C05410=1188.468,337.595,-74.350,-176.324,8.029,148.492
C05411=1188.473,337.346,-74.318,-176.326,8.026,148.492
C05412=1188.477,337.099,-74.285,-176.328,8.022,148.492
C05413=1188.481,336.851,-74.253,-176.331,8.019,148.492
C05414=1188.485,336.602,-74.220,-176.333,8.016,148.491
C05415=1188.489,336.355,-74.189,-176.335,8.014,148.491
C05416=1188.493,336.107,-74.156,-176.337,8.010,148.491
C05417=1188.497,335.859,-74.124,-176.340,8.007,148.491
C05418=1188.502,335.611,-74.091,-176.342,8.004,148.491
C05419=1188.506,335.363,-74.060,-176.344,8.001,148.491
C05420=1188.510,335.116,-74.027,-176.346,7.997,148.490
C05421=1188.514,334.868,-73.995,-176.349,7.994,148.490
C05422=1188.518,334.619,-73.963,-176.351,7.991,148.490
C05423=1188.522,334.372,-73.931,-176.354,7.988,148.490
C05424=1188.526,334.124,-73.899,-176.356,7.985,148.490
C05425=1188.530,333.876,-73.866,-176.358,7.982,148.490
C05426=1188.534,333.628,-73.834,-176.360,7.979,148.490
C05427=1188.539,333.381,-73.802,-176.363,7.976,148.490
C05428=1188.543,333.133,-73.770,-176.365,7.972,148.489
C05429=1188.547,332.884,-73.738,-176.368,7.969,148.489
C05430=1188.552,332.637,-73.706,-176.370,7.966,148.489
C05431=1188.555,332.389,-73.674,-176.372,7.963,148.489
C05432=1188.560,332.140,-73.642,-176.374,7.960,148.489
C05433=1188.563,331.892,-73.610,-176.377,7.957,148.489
C05434=1188.568,331.645,-73.578,-176.379,7.954,148.489
C05435=1188.572,331.397,-73.546,-176.382,7.951,148.489
C05436=1188.576,331.149,-73.514,-176.384,7.948,148.488
C05437=1188.581,330.901,-73.482,-176.386,7.944,148.488
C05438=1188.585,330.653,-73.451,-176.389,7.941,148.488
C05439=1188.588,330.405,-73.419,-176.391,7.938,148.488
C05440=1188.593,330.157,-73.387,-176.394,7.935,148.488
C05441=1188.597,329.909,-73.355,-176.396,7.933,148.488
C05442=1188.601,329.662,-73.323,-176.398,7.929,148.488
C05443=1188.606,329.414,-73.291,-176.401,7.926,148.488
C05444=1188.610,329.166,-73.259,-176.403,7.923,148.487
C05445=1188.614,328.918,-73.228,-176.406,7.920,148.487
C05446=1188.618,328.670,-73.196,-176.408,7.917,148.487
C05447=1188.622,328.421,-73.164,-176.411,7.914,148.487
C05448=1188.627,328.174,-73.132,-176.412,7.911,148.487
C05449=1188.630,327.926,-73.101,-176.414,7.908,148.487
C05450=1188.635,327.678,-73.069,-176.417,7.905,148.487
C05451=1188.639,327.430,-73.037,-176.419,7.901,148.487
C05452=1188.643,327.182,-73.005,-176.422,7.898,148.487
C05453=1188.647,326.934,-72.974,-176.424,7.895,148.486
C05454=1188.651,326.686,-72.942,-176.427,7.892,148.486
C05455=1188.655,326.439,-72.911,-176.429,7.889,148.486
C05456=1188.660,326.190,-72.878,-176.431,7.887,148.486
C05457=1188.664,325.942,-72.847,-176.434,7.883,148.486
C05458=1188.668,325.694,-72.816,-176.436,7.880,148.486
C05459=1188.672,325.446,-72.784,-176.439,7.877,148.486
C05460=1188.676,325.199,-72.752,-176.441,7.874,148.486
C05461=1188.680,324.950,-72.721,-176.444,7.871,148.486
C05462=1188.685,324.703,-72.689,-176.446,7.868,148.486
C05463=1188.689,324.455,-72.657,-176.448,7.865,148.485
C05464=1188.693,324.206,-72.626,-176.451,7.862,148.485
C05465=1188.697,323.959,-72.595,-176.453,7.859,148.485
C05466=1188.701,323.710,-72.564,-176.456,7.856,148.485
C05467=1188.706,323.463,-72.532,-176.458,7.852,148.485
C05468=1188.709,323.215,-72.500,-176.461,7.849,148.485
C05469=1188.714,322.967,-72.470,-176.463,7.846,148.485
C05470=1188.718,322.719,-72.438,-176.465,7.844,148.485
C05471=1188.722,322.471,-72.407,-176.468,7.841,148.485
C05472=1188.727,322.222,-72.374,-176.470,7.838,148.485
C05473=1188.731,321.974,-72.344,-176.473,7.835,148.485
C05474=1188.735,321.726,-72.312,-176.475,7.831,148.484
